   // UNI[6500] := 16#78A3;
   // UNI[6501] := 16#78B2;
   // UNI[6502] := 16#78B9;
   // UNI[6503] := 16#78A5;
   // UNI[6504] := 16#78D4;
   // UNI[6505] := 16#78D9;
   // UNI[6506] := 16#78C9;
   // UNI[6507] := 16#78EC;
   // UNI[6508] := 16#78F2;
   // UNI[6509] := 16#7905;
   // UNI[6510] := 16#78F4;
   // UNI[6511] := 16#7913;
   // UNI[6512] := 16#7924;
   // UNI[6513] := 16#791E;
   // UNI[6514] := 16#7934;
   // UNI[6515] := 16#9F9B;
   // UNI[6516] := 16#9EF9;
   // UNI[6517] := 16#9EFB;
   // UNI[6518] := 16#9EFC;
   // UNI[6519] := 16#76F1;
   // UNI[6520] := 16#7704;
   // UNI[6521] := 16#770D;
   // UNI[6522] := 16#76F9;
   // UNI[6523] := 16#7707;
   // UNI[6524] := 16#7708;
   // UNI[6525] := 16#771A;
   // UNI[6526] := 16#7722;
   // UNI[6527] := 16#7719;
   // UNI[6528] := 16#772D;
   // UNI[6529] := 16#7726;
   // UNI[6530] := 16#7735;
   // UNI[6531] := 16#7738;
   // UNI[6532] := 16#7750;
   // UNI[6533] := 16#7751;
   // UNI[6534] := 16#7747;
   // UNI[6535] := 16#7743;
   // UNI[6536] := 16#775A;
   // UNI[6537] := 16#7768;
   // UNI[6538] := 16#7762;
   // UNI[6539] := 16#7765;
   // UNI[6540] := 16#777F;
   // UNI[6541] := 16#778D;
   // UNI[6542] := 16#777D;
   // UNI[6543] := 16#7780;
   // UNI[6544] := 16#778C;
   // UNI[6545] := 16#7791;
   // UNI[6546] := 16#779F;
   // UNI[6547] := 16#77A0;
   // UNI[6548] := 16#77B0;
   // UNI[6549] := 16#77B5;
   // UNI[6550] := 16#77BD;
   // UNI[6551] := 16#753A;
   // UNI[6552] := 16#7540;
   // UNI[6553] := 16#754E;
   // UNI[6554] := 16#754B;
   // UNI[6555] := 16#7548;
   // UNI[6556] := 16#755B;
   // UNI[6557] := 16#7572;
   // UNI[6558] := 16#7579;
   // UNI[6559] := 16#7583;
   // UNI[6560] := 16#7F58;
   // UNI[6561] := 16#7F61;
   // UNI[6562] := 16#7F5F;
   // UNI[6563] := 16#8A48;
   // UNI[6564] := 16#7F68;
   // UNI[6565] := 16#7F74;
   // UNI[6566] := 16#7F71;
   // UNI[6567] := 16#7F79;
   // UNI[6568] := 16#7F81;
   // UNI[6569] := 16#7F7E;
   // UNI[6570] := 16#76CD;
   // UNI[6571] := 16#76E5;
   // UNI[6572] := 16#8832;
   // UNI[6573] := 16#9485;
   // UNI[6574] := 16#9486;
   // UNI[6575] := 16#9487;
   // UNI[6576] := 16#948B;
   // UNI[6577] := 16#948A;
   // UNI[6578] := 16#948C;
   // UNI[6579] := 16#948D;
   // UNI[6580] := 16#948F;
   // UNI[6581] := 16#9490;
   // UNI[6582] := 16#9494;
   // UNI[6583] := 16#9497;
   // UNI[6584] := 16#9495;
   // UNI[6585] := 16#949A;
   // UNI[6586] := 16#949B;
   // UNI[6587] := 16#949C;
   // UNI[6588] := 16#94A3;
   // UNI[6589] := 16#94A4;
   // UNI[6590] := 16#94AB;
   // UNI[6591] := 16#94AA;
   // UNI[6592] := 16#94AD;
   // UNI[6593] := 16#94AC;
   // UNI[6594] := 16#94AF;
   // UNI[6595] := 16#94B0;
   // UNI[6596] := 16#94B2;
   // UNI[6597] := 16#94B4;
   // UNI[6598] := 16#94B6;
   // UNI[6599] := 16#94B7;
   // UNI[6600] := 16#94B8;
   // UNI[6601] := 16#94B9;
   // UNI[6602] := 16#94BA;
   // UNI[6603] := 16#94BC;
   // UNI[6604] := 16#94BD;
   // UNI[6605] := 16#94BF;
   // UNI[6606] := 16#94C4;
   // UNI[6607] := 16#94C8;
   // UNI[6608] := 16#94C9;
   // UNI[6609] := 16#94CA;
   // UNI[6610] := 16#94CB;
   // UNI[6611] := 16#94CC;
   // UNI[6612] := 16#94CD;
   // UNI[6613] := 16#94CE;
   // UNI[6614] := 16#94D0;
   // UNI[6615] := 16#94D1;
   // UNI[6616] := 16#94D2;
   // UNI[6617] := 16#94D5;
   // UNI[6618] := 16#94D6;
   // UNI[6619] := 16#94D7;
   // UNI[6620] := 16#94D9;
   // UNI[6621] := 16#94D8;
   // UNI[6622] := 16#94DB;
   // UNI[6623] := 16#94DE;
   // UNI[6624] := 16#94DF;
   // UNI[6625] := 16#94E0;
   // UNI[6626] := 16#94E2;
   // UNI[6627] := 16#94E4;
   // UNI[6628] := 16#94E5;
   // UNI[6629] := 16#94E7;
   // UNI[6630] := 16#94E8;
   // UNI[6631] := 16#94EA;
   // UNI[6632] := 16#94E9;
   // UNI[6633] := 16#94EB;
   // UNI[6634] := 16#94EE;
   // UNI[6635] := 16#94EF;
   // UNI[6636] := 16#94F3;
   // UNI[6637] := 16#94F4;
   // UNI[6638] := 16#94F5;
   // UNI[6639] := 16#94F7;
   // UNI[6640] := 16#94F9;
   // UNI[6641] := 16#94FC;
   // UNI[6642] := 16#94FD;
   // UNI[6643] := 16#94FF;
   // UNI[6644] := 16#9503;
   // UNI[6645] := 16#9502;
   // UNI[6646] := 16#9506;
   // UNI[6647] := 16#9507;
   // UNI[6648] := 16#9509;
   // UNI[6649] := 16#950A;
   // UNI[6650] := 16#950D;
   // UNI[6651] := 16#950E;
   // UNI[6652] := 16#950F;
   // UNI[6653] := 16#9512;
   // UNI[6654] := 16#9513;
   // UNI[6655] := 16#9514;
   // UNI[6656] := 16#9515;
   // UNI[6657] := 16#9516;
   // UNI[6658] := 16#9518;
   // UNI[6659] := 16#951B;
   // UNI[6660] := 16#951D;
   // UNI[6661] := 16#951E;
   // UNI[6662] := 16#951F;
   // UNI[6663] := 16#9522;
   // UNI[6664] := 16#952A;
   // UNI[6665] := 16#952B;
   // UNI[6666] := 16#9529;
   // UNI[6667] := 16#952C;
   // UNI[6668] := 16#9531;
   // UNI[6669] := 16#9532;
   // UNI[6670] := 16#9534;
   // UNI[6671] := 16#9536;
   // UNI[6672] := 16#9537;
   // UNI[6673] := 16#9538;
   // UNI[6674] := 16#953C;
   // UNI[6675] := 16#953E;
   // UNI[6676] := 16#953F;
   // UNI[6677] := 16#9542;
   // UNI[6678] := 16#9535;
   // UNI[6679] := 16#9544;
   // UNI[6680] := 16#9545;
   // UNI[6681] := 16#9546;
   // UNI[6682] := 16#9549;
   // UNI[6683] := 16#954C;
   // UNI[6684] := 16#954E;
   // UNI[6685] := 16#954F;
   // UNI[6686] := 16#9552;
   // UNI[6687] := 16#9553;
   // UNI[6688] := 16#9554;
   // UNI[6689] := 16#9556;
   // UNI[6690] := 16#9557;
   // UNI[6691] := 16#9558;
   // UNI[6692] := 16#9559;
   // UNI[6693] := 16#955B;
   // UNI[6694] := 16#955E;
   // UNI[6695] := 16#955F;
   // UNI[6696] := 16#955D;
   // UNI[6697] := 16#9561;
   // UNI[6698] := 16#9562;
   // UNI[6699] := 16#9564;
   // UNI[6700] := 16#9565;
   // UNI[6701] := 16#9566;
   // UNI[6702] := 16#9567;
   // UNI[6703] := 16#9568;
   // UNI[6704] := 16#9569;
   // UNI[6705] := 16#956A;
   // UNI[6706] := 16#956B;
   // UNI[6707] := 16#956C;
   // UNI[6708] := 16#956F;
   // UNI[6709] := 16#9571;
   // UNI[6710] := 16#9572;
   // UNI[6711] := 16#9573;
   // UNI[6712] := 16#953A;
   // UNI[6713] := 16#77E7;
   // UNI[6714] := 16#77EC;
   // UNI[6715] := 16#96C9;
   // UNI[6716] := 16#79D5;
   // UNI[6717] := 16#79ED;
   // UNI[6718] := 16#79E3;
   // UNI[6719] := 16#79EB;
   // UNI[6720] := 16#7A06;
   // UNI[6721] := 16#5D47;
   // UNI[6722] := 16#7A03;
   // UNI[6723] := 16#7A02;
   // UNI[6724] := 16#7A1E;
   // UNI[6725] := 16#7A14;
   // UNI[6726] := 16#7A39;
   // UNI[6727] := 16#7A37;
   // UNI[6728] := 16#7A51;
   // UNI[6729] := 16#9ECF;
   // UNI[6730] := 16#99A5;
   // UNI[6731] := 16#7A70;
   // UNI[6732] := 16#7688;
   // UNI[6733] := 16#768E;
   // UNI[6734] := 16#7693;
   // UNI[6735] := 16#7699;
   // UNI[6736] := 16#76A4;
   // UNI[6737] := 16#74DE;
   // UNI[6738] := 16#74E0;
   // UNI[6739] := 16#752C;
   // UNI[6740] := 16#9E20;
   // UNI[6741] := 16#9E22;
   // UNI[6742] := 16#9E28;
   // UNI[6743] := 16#9E29;
   // UNI[6744] := 16#9E2A;
   // UNI[6745] := 16#9E2B;
   // UNI[6746] := 16#9E2C;
   // UNI[6747] := 16#9E32;
   // UNI[6748] := 16#9E31;
   // UNI[6749] := 16#9E36;
   // UNI[6750] := 16#9E38;
   // UNI[6751] := 16#9E37;
   // UNI[6752] := 16#9E39;
   // UNI[6753] := 16#9E3A;
   // UNI[6754] := 16#9E3E;
   // UNI[6755] := 16#9E41;
   // UNI[6756] := 16#9E42;
   // UNI[6757] := 16#9E44;
   // UNI[6758] := 16#9E46;
   // UNI[6759] := 16#9E47;
   // UNI[6760] := 16#9E48;
   // UNI[6761] := 16#9E49;
   // UNI[6762] := 16#9E4B;
   // UNI[6763] := 16#9E4C;
   // UNI[6764] := 16#9E4E;
   // UNI[6765] := 16#9E51;
   // UNI[6766] := 16#9E55;
   // UNI[6767] := 16#9E57;
   // UNI[6768] := 16#9E5A;
   // UNI[6769] := 16#9E5B;
   // UNI[6770] := 16#9E5C;
   // UNI[6771] := 16#9E5E;
   // UNI[6772] := 16#9E63;
   // UNI[6773] := 16#9E66;
   // UNI[6774] := 16#9E67;
   // UNI[6775] := 16#9E68;
   // UNI[6776] := 16#9E69;
   // UNI[6777] := 16#9E6A;
   // UNI[6778] := 16#9E6B;
   // UNI[6779] := 16#9E6C;
   // UNI[6780] := 16#9E71;
   // UNI[6781] := 16#9E6D;
   // UNI[6782] := 16#9E73;
   // UNI[6783] := 16#7592;
   // UNI[6784] := 16#7594;
   // UNI[6785] := 16#7596;
   // UNI[6786] := 16#75A0;
   // UNI[6787] := 16#759D;
   // UNI[6788] := 16#75AC;
   // UNI[6789] := 16#75A3;
   // UNI[6790] := 16#75B3;
   // UNI[6791] := 16#75B4;
   // UNI[6792] := 16#75B8;
   // UNI[6793] := 16#75C4;
   // UNI[6794] := 16#75B1;
   // UNI[6795] := 16#75B0;
   // UNI[6796] := 16#75C3;
   // UNI[6797] := 16#75C2;
   // UNI[6798] := 16#75D6;
   // UNI[6799] := 16#75CD;
   // UNI[6800] := 16#75E3;
   // UNI[6801] := 16#75E8;
   // UNI[6802] := 16#75E6;
   // UNI[6803] := 16#75E4;
   // UNI[6804] := 16#75EB;
   // UNI[6805] := 16#75E7;
   // UNI[6806] := 16#7603;
   // UNI[6807] := 16#75F1;
   // UNI[6808] := 16#75FC;
   // UNI[6809] := 16#75FF;
   // UNI[6810] := 16#7610;
   // UNI[6811] := 16#7600;
   // UNI[6812] := 16#7605;
   // UNI[6813] := 16#760C;
   // UNI[6814] := 16#7617;
   // UNI[6815] := 16#760A;
   // UNI[6816] := 16#7625;
   // UNI[6817] := 16#7618;
   // UNI[6818] := 16#7615;
   // UNI[6819] := 16#7619;
   // UNI[6820] := 16#761B;
   // UNI[6821] := 16#763C;
   // UNI[6822] := 16#7622;
   // UNI[6823] := 16#7620;
   // UNI[6824] := 16#7640;
   // UNI[6825] := 16#762D;
   // UNI[6826] := 16#7630;
   // UNI[6827] := 16#763F;
   // UNI[6828] := 16#7635;
   // UNI[6829] := 16#7643;
   // UNI[6830] := 16#763E;
   // UNI[6831] := 16#7633;
   // UNI[6832] := 16#764D;
   // UNI[6833] := 16#765E;
   // UNI[6834] := 16#7654;
   // UNI[6835] := 16#765C;
   // UNI[6836] := 16#7656;
   // UNI[6837] := 16#766B;
   // UNI[6838] := 16#766F;
   // UNI[6839] := 16#7FCA;
   // UNI[6840] := 16#7AE6;
   // UNI[6841] := 16#7A78;
   // UNI[6842] := 16#7A79;
   // UNI[6843] := 16#7A80;
   // UNI[6844] := 16#7A86;
   // UNI[6845] := 16#7A88;
   // UNI[6846] := 16#7A95;
   // UNI[6847] := 16#7AA6;
   // UNI[6848] := 16#7AA0;
   // UNI[6849] := 16#7AAC;
   // UNI[6850] := 16#7AA8;
   // UNI[6851] := 16#7AAD;
   // UNI[6852] := 16#7AB3;
   // UNI[6853] := 16#8864;
   // UNI[6854] := 16#8869;
   // UNI[6855] := 16#8872;
   // UNI[6856] := 16#887D;
   // UNI[6857] := 16#887F;
   // UNI[6858] := 16#8882;
   // UNI[6859] := 16#88A2;
   // UNI[6860] := 16#88C6;
   // UNI[6861] := 16#88B7;
   // UNI[6862] := 16#88BC;
   // UNI[6863] := 16#88C9;
   // UNI[6864] := 16#88E2;
   // UNI[6865] := 16#88CE;
   // UNI[6866] := 16#88E3;
   // UNI[6867] := 16#88E5;
   // UNI[6868] := 16#88F1;
   // UNI[6869] := 16#891A;
   // UNI[6870] := 16#88FC;
   // UNI[6871] := 16#88E8;
   // UNI[6872] := 16#88FE;
   // UNI[6873] := 16#88F0;
   // UNI[6874] := 16#8921;
   // UNI[6875] := 16#8919;
   // UNI[6876] := 16#8913;
   // UNI[6877] := 16#891B;
   // UNI[6878] := 16#890A;
   // UNI[6879] := 16#8934;
   // UNI[6880] := 16#892B;
   // UNI[6881] := 16#8936;
   // UNI[6882] := 16#8941;
   // UNI[6883] := 16#8966;
   // UNI[6884] := 16#897B;
   // UNI[6885] := 16#758B;
   // UNI[6886] := 16#80E5;
   // UNI[6887] := 16#76B2;
   // UNI[6888] := 16#76B4;
   // UNI[6889] := 16#77DC;
   // UNI[6890] := 16#8012;
   // UNI[6891] := 16#8014;
   // UNI[6892] := 16#8016;
   // UNI[6893] := 16#801C;
   // UNI[6894] := 16#8020;
   // UNI[6895] := 16#8022;
   // UNI[6896] := 16#8025;
   // UNI[6897] := 16#8026;
   // UNI[6898] := 16#8027;
   // UNI[6899] := 16#8029;
   // UNI[6900] := 16#8028;
   // UNI[6901] := 16#8031;
   // UNI[6902] := 16#800B;
   // UNI[6903] := 16#8035;
   // UNI[6904] := 16#8043;
   // UNI[6905] := 16#8046;
   // UNI[6906] := 16#804D;
   // UNI[6907] := 16#8052;
   // UNI[6908] := 16#8069;
   // UNI[6909] := 16#8071;
   // UNI[6910] := 16#8983;
   // UNI[6911] := 16#9878;
   // UNI[6912] := 16#9880;
   // UNI[6913] := 16#9883;
   // UNI[6914] := 16#9889;
   // UNI[6915] := 16#988C;
   // UNI[6916] := 16#988D;
   // UNI[6917] := 16#988F;
   // UNI[6918] := 16#9894;
   // UNI[6919] := 16#989A;
   // UNI[6920] := 16#989B;
   // UNI[6921] := 16#989E;
   // UNI[6922] := 16#989F;
   // UNI[6923] := 16#98A1;
   // UNI[6924] := 16#98A2;
   // UNI[6925] := 16#98A5;
   // UNI[6926] := 16#98A6;
   // UNI[6927] := 16#864D;
   // UNI[6928] := 16#8654;
   // UNI[6929] := 16#866C;
   // UNI[6930] := 16#866E;
   // UNI[6931] := 16#867F;
   // UNI[6932] := 16#867A;
   // UNI[6933] := 16#867C;
   // UNI[6934] := 16#867B;
   // UNI[6935] := 16#86A8;
   // UNI[6936] := 16#868D;
   // UNI[6937] := 16#868B;
   // UNI[6938] := 16#86AC;
   // UNI[6939] := 16#869D;
   // UNI[6940] := 16#86A7;
   // UNI[6941] := 16#86A3;
   // UNI[6942] := 16#86AA;
   // UNI[6943] := 16#8693;
   // UNI[6944] := 16#86A9;
   // UNI[6945] := 16#86B6;
   // UNI[6946] := 16#86C4;
   // UNI[6947] := 16#86B5;
   // UNI[6948] := 16#86CE;
   // UNI[6949] := 16#86B0;
   // UNI[6950] := 16#86BA;
   // UNI[6951] := 16#86B1;
   // UNI[6952] := 16#86AF;
   // UNI[6953] := 16#86C9;
   // UNI[6954] := 16#86CF;
   // UNI[6955] := 16#86B4;
   // UNI[6956] := 16#86E9;
   // UNI[6957] := 16#86F1;
   // UNI[6958] := 16#86F2;
   // UNI[6959] := 16#86ED;
   // UNI[6960] := 16#86F3;
   // UNI[6961] := 16#86D0;
   // UNI[6962] := 16#8713;
   // UNI[6963] := 16#86DE;
   // UNI[6964] := 16#86F4;
   // UNI[6965] := 16#86DF;
   // UNI[6966] := 16#86D8;
   // UNI[6967] := 16#86D1;
   // UNI[6968] := 16#8703;
   // UNI[6969] := 16#8707;
   // UNI[6970] := 16#86F8;
   // UNI[6971] := 16#8708;
   // UNI[6972] := 16#870A;
   // UNI[6973] := 16#870D;
   // UNI[6974] := 16#8709;
   // UNI[6975] := 16#8723;
   // UNI[6976] := 16#873B;
   // UNI[6977] := 16#871E;
   // UNI[6978] := 16#8725;
   // UNI[6979] := 16#872E;
   // UNI[6980] := 16#871A;
   // UNI[6981] := 16#873E;
   // UNI[6982] := 16#8748;
   // UNI[6983] := 16#8734;
   // UNI[6984] := 16#8731;
   // UNI[6985] := 16#8729;
   // UNI[6986] := 16#8737;
   // UNI[6987] := 16#873F;
   // UNI[6988] := 16#8782;
   // UNI[6989] := 16#8722;
   // UNI[6990] := 16#877D;
   // UNI[6991] := 16#877E;
   // UNI[6992] := 16#877B;
   // UNI[6993] := 16#8760;
   // UNI[6994] := 16#8770;
   // UNI[6995] := 16#874C;
   // UNI[6996] := 16#876E;
   // UNI[6997] := 16#878B;
   // UNI[6998] := 16#8753;
   // UNI[6999] := 16#8763;
   // UNI[7000] := 16#877C;
   // UNI[7001] := 16#8764;
   // UNI[7002] := 16#8759;
   // UNI[7003] := 16#8765;
   // UNI[7004] := 16#8793;
   // UNI[7005] := 16#87AF;
   // UNI[7006] := 16#87A8;
   // UNI[7007] := 16#87D2;
   // UNI[7008] := 16#87C6;
   // UNI[7009] := 16#8788;
   // UNI[7010] := 16#8785;
   // UNI[7011] := 16#87AD;
   // UNI[7012] := 16#8797;
   // UNI[7013] := 16#8783;
   // UNI[7014] := 16#87AB;
   // UNI[7015] := 16#87E5;
   // UNI[7016] := 16#87AC;
   // UNI[7017] := 16#87B5;
   // UNI[7018] := 16#87B3;
   // UNI[7019] := 16#87CB;
   // UNI[7020] := 16#87D3;
   // UNI[7021] := 16#87BD;
   // UNI[7022] := 16#87D1;
   // UNI[7023] := 16#87C0;
   // UNI[7024] := 16#87CA;
   // UNI[7025] := 16#87DB;
   // UNI[7026] := 16#87EA;
   // UNI[7027] := 16#87E0;
   // UNI[7028] := 16#87EE;
   // UNI[7029] := 16#8816;
   // UNI[7030] := 16#8813;
   // UNI[7031] := 16#87FE;
   // UNI[7032] := 16#880A;
   // UNI[7033] := 16#881B;
   // UNI[7034] := 16#8821;
   // UNI[7035] := 16#8839;
   // UNI[7036] := 16#883C;
   // UNI[7037] := 16#7F36;
   // UNI[7038] := 16#7F42;
   // UNI[7039] := 16#7F44;
   // UNI[7040] := 16#7F45;
   // UNI[7041] := 16#8210;
   // UNI[7042] := 16#7AFA;
   // UNI[7043] := 16#7AFD;
   // UNI[7044] := 16#7B08;
   // UNI[7045] := 16#7B03;
   // UNI[7046] := 16#7B04;
   // UNI[7047] := 16#7B15;
   // UNI[7048] := 16#7B0A;
   // UNI[7049] := 16#7B2B;
   // UNI[7050] := 16#7B0F;
   // UNI[7051] := 16#7B47;
   // UNI[7052] := 16#7B38;
   // UNI[7053] := 16#7B2A;
   // UNI[7054] := 16#7B19;
   // UNI[7055] := 16#7B2E;
   // UNI[7056] := 16#7B31;
   // UNI[7057] := 16#7B20;
   // UNI[7058] := 16#7B25;
   // UNI[7059] := 16#7B24;
   // UNI[7060] := 16#7B33;
   // UNI[7061] := 16#7B3E;
   // UNI[7062] := 16#7B1E;
   // UNI[7063] := 16#7B58;
   // UNI[7064] := 16#7B5A;
   // UNI[7065] := 16#7B45;
   // UNI[7066] := 16#7B75;
   // UNI[7067] := 16#7B4C;
   // UNI[7068] := 16#7B5D;
   // UNI[7069] := 16#7B60;
   // UNI[7070] := 16#7B6E;
   // UNI[7071] := 16#7B7B;
   // UNI[7072] := 16#7B62;
   // UNI[7073] := 16#7B72;
   // UNI[7074] := 16#7B71;
   // UNI[7075] := 16#7B90;
   // UNI[7076] := 16#7BA6;
   // UNI[7077] := 16#7BA7;
   // UNI[7078] := 16#7BB8;
   // UNI[7079] := 16#7BAC;
   // UNI[7080] := 16#7B9D;
   // UNI[7081] := 16#7BA8;
   // UNI[7082] := 16#7B85;
   // UNI[7083] := 16#7BAA;
   // UNI[7084] := 16#7B9C;
   // UNI[7085] := 16#7BA2;
   // UNI[7086] := 16#7BAB;
   // UNI[7087] := 16#7BB4;
   // UNI[7088] := 16#7BD1;
   // UNI[7089] := 16#7BC1;
   // UNI[7090] := 16#7BCC;
   // UNI[7091] := 16#7BDD;
   // UNI[7092] := 16#7BDA;
   // UNI[7093] := 16#7BE5;
   // UNI[7094] := 16#7BE6;
   // UNI[7095] := 16#7BEA;
   // UNI[7096] := 16#7C0C;
   // UNI[7097] := 16#7BFE;
   // UNI[7098] := 16#7BFC;
   // UNI[7099] := 16#7C0F;
   // UNI[7100] := 16#7C16;
   // UNI[7101] := 16#7C0B;
   // UNI[7102] := 16#7C1F;
   // UNI[7103] := 16#7C2A;
   // UNI[7104] := 16#7C26;
   // UNI[7105] := 16#7C38;
   // UNI[7106] := 16#7C41;
   // UNI[7107] := 16#7C40;
   // UNI[7108] := 16#81FE;
   // UNI[7109] := 16#8201;
   // UNI[7110] := 16#8202;
   // UNI[7111] := 16#8204;
   // UNI[7112] := 16#81EC;
   // UNI[7113] := 16#8844;
   // UNI[7114] := 16#8221;
   // UNI[7115] := 16#8222;
   // UNI[7116] := 16#8223;
   // UNI[7117] := 16#822D;
   // UNI[7118] := 16#822F;
   // UNI[7119] := 16#8228;
   // UNI[7120] := 16#822B;
   // UNI[7121] := 16#8238;
   // UNI[7122] := 16#823B;
   // UNI[7123] := 16#8233;
   // UNI[7124] := 16#8234;
   // UNI[7125] := 16#823E;
   // UNI[7126] := 16#8244;
   // UNI[7127] := 16#8249;
   // UNI[7128] := 16#824B;
   // UNI[7129] := 16#824F;
   // UNI[7130] := 16#825A;
   // UNI[7131] := 16#825F;
   // UNI[7132] := 16#8268;
   // UNI[7133] := 16#887E;
   // UNI[7134] := 16#8885;
   // UNI[7135] := 16#8888;
   // UNI[7136] := 16#88D8;
   // UNI[7137] := 16#88DF;
   // UNI[7138] := 16#895E;
   // UNI[7139] := 16#7F9D;
   // UNI[7140] := 16#7F9F;
   // UNI[7141] := 16#7FA7;
   // UNI[7142] := 16#7FAF;
   // UNI[7143] := 16#7FB0;
   // UNI[7144] := 16#7FB2;
   // UNI[7145] := 16#7C7C;
   // UNI[7146] := 16#6549;
   // UNI[7147] := 16#7C91;
   // UNI[7148] := 16#7C9D;
   // UNI[7149] := 16#7C9C;
   // UNI[7150] := 16#7C9E;
   // UNI[7151] := 16#7CA2;
   // UNI[7152] := 16#7CB2;
   // UNI[7153] := 16#7CBC;
   // UNI[7154] := 16#7CBD;
   // UNI[7155] := 16#7CC1;
   // UNI[7156] := 16#7CC7;
   // UNI[7157] := 16#7CCC;
   // UNI[7158] := 16#7CCD;
   // UNI[7159] := 16#7CC8;
   // UNI[7160] := 16#7CC5;
   // UNI[7161] := 16#7CD7;
   // UNI[7162] := 16#7CE8;
   // UNI[7163] := 16#826E;
   // UNI[7164] := 16#66A8;
   // UNI[7165] := 16#7FBF;
   // UNI[7166] := 16#7FCE;
   // UNI[7167] := 16#7FD5;
   // UNI[7168] := 16#7FE5;
   // UNI[7169] := 16#7FE1;
   // UNI[7170] := 16#7FE6;
   // UNI[7171] := 16#7FE9;
   // UNI[7172] := 16#7FEE;
   // UNI[7173] := 16#7FF3;
   // UNI[7174] := 16#7CF8;
   // UNI[7175] := 16#7D77;
   // UNI[7176] := 16#7DA6;
   // UNI[7177] := 16#7DAE;
   // UNI[7178] := 16#7E47;
   // UNI[7179] := 16#7E9B;
   // UNI[7180] := 16#9EB8;
   // UNI[7181] := 16#9EB4;
   // UNI[7182] := 16#8D73;
   // UNI[7183] := 16#8D84;
   // UNI[7184] := 16#8D94;
   // UNI[7185] := 16#8D91;
   // UNI[7186] := 16#8DB1;
   // UNI[7187] := 16#8D67;
   // UNI[7188] := 16#8D6D;
   // UNI[7189] := 16#8C47;
   // UNI[7190] := 16#8C49;
   // UNI[7191] := 16#914A;
   // UNI[7192] := 16#9150;
   // UNI[7193] := 16#914E;
   // UNI[7194] := 16#914F;
   // UNI[7195] := 16#9164;
   // UNI[7196] := 16#9162;
   // UNI[7197] := 16#9161;
   // UNI[7198] := 16#9170;
   // UNI[7199] := 16#9169;
   // UNI[7200] := 16#916F;
   // UNI[7201] := 16#917D;
   // UNI[7202] := 16#917E;
   // UNI[7203] := 16#9172;
   // UNI[7204] := 16#9174;
   // UNI[7205] := 16#9179;
   // UNI[7206] := 16#918C;
   // UNI[7207] := 16#9185;
   // UNI[7208] := 16#9190;
   // UNI[7209] := 16#918D;
   // UNI[7210] := 16#9191;
   // UNI[7211] := 16#91A2;
   // UNI[7212] := 16#91A3;
   // UNI[7213] := 16#91AA;
   // UNI[7214] := 16#91AD;
   // UNI[7215] := 16#91AE;
   // UNI[7216] := 16#91AF;
   // UNI[7217] := 16#91B5;
   // UNI[7218] := 16#91B4;
   // UNI[7219] := 16#91BA;
   // UNI[7220] := 16#8C55;
   // UNI[7221] := 16#9E7E;
   // UNI[7222] := 16#8DB8;
   // UNI[7223] := 16#8DEB;
   // UNI[7224] := 16#8E05;
   // UNI[7225] := 16#8E59;
   // UNI[7226] := 16#8E69;
   // UNI[7227] := 16#8DB5;
   // UNI[7228] := 16#8DBF;
   // UNI[7229] := 16#8DBC;
   // UNI[7230] := 16#8DBA;
   // UNI[7231] := 16#8DC4;
   // UNI[7232] := 16#8DD6;
   // UNI[7233] := 16#8DD7;
   // UNI[7234] := 16#8DDA;
   // UNI[7235] := 16#8DDE;
   // UNI[7236] := 16#8DCE;
   // UNI[7237] := 16#8DCF;
   // UNI[7238] := 16#8DDB;
   // UNI[7239] := 16#8DC6;
   // UNI[7240] := 16#8DEC;
   // UNI[7241] := 16#8DF7;
   // UNI[7242] := 16#8DF8;
   // UNI[7243] := 16#8DE3;
   // UNI[7244] := 16#8DF9;
   // UNI[7245] := 16#8DFB;
   // UNI[7246] := 16#8DE4;
   // UNI[7247] := 16#8E09;
   // UNI[7248] := 16#8DFD;
   // UNI[7249] := 16#8E14;
   // UNI[7250] := 16#8E1D;
   // UNI[7251] := 16#8E1F;
   // UNI[7252] := 16#8E2C;
   // UNI[7253] := 16#8E2E;
   // UNI[7254] := 16#8E23;
   // UNI[7255] := 16#8E2F;
   // UNI[7256] := 16#8E3A;
   // UNI[7257] := 16#8E40;
   // UNI[7258] := 16#8E39;
   // UNI[7259] := 16#8E35;
   // UNI[7260] := 16#8E3D;
   // UNI[7261] := 16#8E31;
   // UNI[7262] := 16#8E49;
   // UNI[7263] := 16#8E41;
   // UNI[7264] := 16#8E42;
   // UNI[7265] := 16#8E51;
   // UNI[7266] := 16#8E52;
   // UNI[7267] := 16#8E4A;
   // UNI[7268] := 16#8E70;
   // UNI[7269] := 16#8E76;
   // UNI[7270] := 16#8E7C;
   // UNI[7271] := 16#8E6F;
   // UNI[7272] := 16#8E74;
   // UNI[7273] := 16#8E85;
   // UNI[7274] := 16#8E8F;
   // UNI[7275] := 16#8E94;
   // UNI[7276] := 16#8E90;
   // UNI[7277] := 16#8E9C;
   // UNI[7278] := 16#8E9E;
   // UNI[7279] := 16#8C78;
   // UNI[7280] := 16#8C82;
   // UNI[7281] := 16#8C8A;
   // UNI[7282] := 16#8C85;
   // UNI[7283] := 16#8C98;
   // UNI[7284] := 16#8C94;
   // UNI[7285] := 16#659B;
   // UNI[7286] := 16#89D6;
   // UNI[7287] := 16#89DE;
   // UNI[7288] := 16#89DA;
   // UNI[7289] := 16#89DC;
   // UNI[7290] := 16#89E5;
   // UNI[7291] := 16#89EB;
   // UNI[7292] := 16#89EF;
   // UNI[7293] := 16#8A3E;
   // UNI[7294] := 16#8B26;
   // UNI[7295] := 16#9753;
   // UNI[7296] := 16#96E9;
   // UNI[7297] := 16#96F3;
   // UNI[7298] := 16#96EF;
   // UNI[7299] := 16#9706;
   // UNI[7300] := 16#9701;
   // UNI[7301] := 16#9708;
   // UNI[7302] := 16#970F;
   // UNI[7303] := 16#970E;
   // UNI[7304] := 16#972A;
   // UNI[7305] := 16#972D;
   // UNI[7306] := 16#9730;
   // UNI[7307] := 16#973E;
   // UNI[7308] := 16#9F80;
   // UNI[7309] := 16#9F83;
   // UNI[7310] := 16#9F85;
   // UNI[7311] := 16#9F86;
   // UNI[7312] := 16#9F87;
   // UNI[7313] := 16#9F88;
   // UNI[7314] := 16#9F89;
   // UNI[7315] := 16#9F8A;
   // UNI[7316] := 16#9F8C;
   // UNI[7317] := 16#9EFE;
   // UNI[7318] := 16#9F0B;
   // UNI[7319] := 16#9F0D;
   // UNI[7320] := 16#96B9;
   // UNI[7321] := 16#96BC;
   // UNI[7322] := 16#96BD;
   // UNI[7323] := 16#96CE;
   // UNI[7324] := 16#96D2;
   // UNI[7325] := 16#77BF;
   // UNI[7326] := 16#96E0;
   // UNI[7327] := 16#928E;
   // UNI[7328] := 16#92AE;
   // UNI[7329] := 16#92C8;
   // UNI[7330] := 16#933E;
   // UNI[7331] := 16#936A;
   // UNI[7332] := 16#93CA;
   // UNI[7333] := 16#938F;
   // UNI[7334] := 16#943E;
   // UNI[7335] := 16#946B;
   // UNI[7336] := 16#9C7F;
   // UNI[7337] := 16#9C82;
   // UNI[7338] := 16#9C85;
   // UNI[7339] := 16#9C86;
   // UNI[7340] := 16#9C87;
   // UNI[7341] := 16#9C88;
   // UNI[7342] := 16#7A23;
   // UNI[7343] := 16#9C8B;
   // UNI[7344] := 16#9C8E;
   // UNI[7345] := 16#9C90;
   // UNI[7346] := 16#9C91;
   // UNI[7347] := 16#9C92;
   // UNI[7348] := 16#9C94;
   // UNI[7349] := 16#9C95;
   // UNI[7350] := 16#9C9A;
   // UNI[7351] := 16#9C9B;
   // UNI[7352] := 16#9C9E;
   // UNI[7353] := 16#9C9F;
   // UNI[7354] := 16#9CA0;
   // UNI[7355] := 16#9CA1;
   // UNI[7356] := 16#9CA2;
   // UNI[7357] := 16#9CA3;
   // UNI[7358] := 16#9CA5;
   // UNI[7359] := 16#9CA6;
   // UNI[7360] := 16#9CA7;
   // UNI[7361] := 16#9CA8;
   // UNI[7362] := 16#9CA9;
   // UNI[7363] := 16#9CAB;
   // UNI[7364] := 16#9CAD;
   // UNI[7365] := 16#9CAE;
   // UNI[7366] := 16#9CB0;
   // UNI[7367] := 16#9CB1;
   // UNI[7368] := 16#9CB2;
   // UNI[7369] := 16#9CB3;
   // UNI[7370] := 16#9CB4;
   // UNI[7371] := 16#9CB5;
   // UNI[7372] := 16#9CB6;
   // UNI[7373] := 16#9CB7;
   // UNI[7374] := 16#9CBA;
   // UNI[7375] := 16#9CBB;
   // UNI[7376] := 16#9CBC;
   // UNI[7377] := 16#9CBD;
   // UNI[7378] := 16#9CC4;
   // UNI[7379] := 16#9CC5;
   // UNI[7380] := 16#9CC6;
   // UNI[7381] := 16#9CC7;
   // UNI[7382] := 16#9CCA;
   // UNI[7383] := 16#9CCB;
   // UNI[7384] := 16#9CCC;
   // UNI[7385] := 16#9CCD;
   // UNI[7386] := 16#9CCE;
   // UNI[7387] := 16#9CCF;
   // UNI[7388] := 16#9CD0;
   // UNI[7389] := 16#9CD3;
   // UNI[7390] := 16#9CD4;
   // UNI[7391] := 16#9CD5;
   // UNI[7392] := 16#9CD7;
   // UNI[7393] := 16#9CD8;
   // UNI[7394] := 16#9CD9;
   // UNI[7395] := 16#9CDC;
   // UNI[7396] := 16#9CDD;
   // UNI[7397] := 16#9CDF;
   // UNI[7398] := 16#9CE2;
   // UNI[7399] := 16#977C;
   // UNI[7400] := 16#9785;
   // UNI[7401] := 16#9791;
   // UNI[7402] := 16#9792;
   // UNI[7403] := 16#9794;
   // UNI[7404] := 16#97AF;
   // UNI[7405] := 16#97AB;
   // UNI[7406] := 16#97A3;
   // UNI[7407] := 16#97B2;
   // UNI[7408] := 16#97B4;
   // UNI[7409] := 16#9AB1;
   // UNI[7410] := 16#9AB0;
   // UNI[7411] := 16#9AB7;
   // UNI[7412] := 16#9E58;
   // UNI[7413] := 16#9AB6;
   // UNI[7414] := 16#9ABA;
   // UNI[7415] := 16#9ABC;
   // UNI[7416] := 16#9AC1;
   // UNI[7417] := 16#9AC0;
   // UNI[7418] := 16#9AC5;
   // UNI[7419] := 16#9AC2;
   // UNI[7420] := 16#9ACB;
   // UNI[7421] := 16#9ACC;
   // UNI[7422] := 16#9AD1;
   // UNI[7423] := 16#9B45;
   // UNI[7424] := 16#9B43;
   // UNI[7425] := 16#9B47;
   // UNI[7426] := 16#9B49;
   // UNI[7427] := 16#9B48;
   // UNI[7428] := 16#9B4D;
   // UNI[7429] := 16#9B51;
   // UNI[7430] := 16#98E8;
   // UNI[7431] := 16#990D;
   // UNI[7432] := 16#992E;
   // UNI[7433] := 16#9955;
   // UNI[7434] := 16#9954;
   // UNI[7435] := 16#9ADF;
   // UNI[7436] := 16#9AE1;
   // UNI[7437] := 16#9AE6;
   // UNI[7438] := 16#9AEF;
   // UNI[7439] := 16#9AEB;
   // UNI[7440] := 16#9AFB;
   // UNI[7441] := 16#9AED;
   // UNI[7442] := 16#9AF9;
   // UNI[7443] := 16#9B08;
   // UNI[7444] := 16#9B0F;
   // UNI[7445] := 16#9B13;
   // UNI[7446] := 16#9B1F;
   // UNI[7447] := 16#9B23;
   // UNI[7448] := 16#9EBD;
   // UNI[7449] := 16#9EBE;
   // UNI[7450] := 16#7E3B;
   // UNI[7451] := 16#9E82;
   // UNI[7452] := 16#9E87;
   // UNI[7453] := 16#9E88;
   // UNI[7454] := 16#9E8B;
   // UNI[7455] := 16#9E92;
   // UNI[7456] := 16#93D6;
   // UNI[7457] := 16#9E9D;
   // UNI[7458] := 16#9E9F;
   // UNI[7459] := 16#9EDB;
   // UNI[7460] := 16#9EDC;
   // UNI[7461] := 16#9EDD;
   // UNI[7462] := 16#9EE0;
   // UNI[7463] := 16#9EDF;
   // UNI[7464] := 16#9EE2;
   // UNI[7465] := 16#9EE9;
   // UNI[7466] := 16#9EE7;
   // UNI[7467] := 16#9EE5;
   // UNI[7468] := 16#9EEA;
   // UNI[7469] := 16#9EEF;
   // UNI[7470] := 16#9F22;
   // UNI[7471] := 16#9F2C;
   // UNI[7472] := 16#9F2F;
   // UNI[7473] := 16#9F39;
   // UNI[7474] := 16#9F37;
   // UNI[7475] := 16#9F3D;
   // UNI[7476] := 16#9F3E;
   // UNI[7477] := 16#9F44;
   // UNI[7478] := 0;
   // UNI[7479] := 0;
BEGIN
   IF #GB2312 < 16#0080 THEN
       #UNICODE := #GB2312;
   ELSE
       #hi := 7480;
       #li := 0;
       FOR #j := 0 TO 13 BY 1 DO
           #i := #li + (#hi - #li) / 2;
           IF #GB2312 = #GB2[#i] THEN
               #UNICODE := #UNI[#i];
               EXIT;
           END_IF;
           IF #GB2312 > #GB2[#i] THEN
               #li := #i;
           ELSE
               #hi := #i;
           END_IF;
       END_FOR;
   END_IF;
END_FUNCTION_BLOCK

// ===== library: MasterCopy "GBK_TO_UNI" =====

// folder: FB/UNICODE_FB

FUNCTION_BLOCK "GBK_TO_UNI"   // FB2, SCL
{ S7_Optimized_Access := 'TRUE' }
VERSION : 0.1
   VAR_INPUT
      GBK : Word;
   END_VAR
   VAR_OUTPUT
      UNICODE : Word;
   END_VAR
   VAR
      GBK_TO_UNICODE : Array[0..43592] of Word;
   END_VAR
   VAR_TEMP
      i : UDInt;
      j : UDInt;
      li : UDInt;
      hi : UDInt;
   END_VAR
   // GBK_TO_UNICODE[0] := 16#0080;
   // GBK_TO_UNICODE[1] := 16#20AC;
   // GBK_TO_UNICODE[2] := 16#8140;
   // GBK_TO_UNICODE[3] := 16#4E02;
   // GBK_TO_UNICODE[4] := 16#8141;
   // GBK_TO_UNICODE[5] := 16#4E04;
   // GBK_TO_UNICODE[6] := 16#8142;
   // GBK_TO_UNICODE[7] := 16#4E05;
   // GBK_TO_UNICODE[8] := 16#8143;
   // GBK_TO_UNICODE[9] := 16#4E06;
   // GBK_TO_UNICODE[10] := 16#8144;
   // GBK_TO_UNICODE[11] := 16#4E0F;
   // GBK_TO_UNICODE[12] := 16#8145;
   // GBK_TO_UNICODE[13] := 16#4E12;
   // GBK_TO_UNICODE[14] := 16#8146;
   // GBK_TO_UNICODE[15] := 16#4E17;
   // GBK_TO_UNICODE[16] := 16#8147;
   // GBK_TO_UNICODE[17] := 16#4E1F;
   // GBK_TO_UNICODE[18] := 16#8148;
   // GBK_TO_UNICODE[19] := 16#4E20;
   // GBK_TO_UNICODE[20] := 16#8149;
   // GBK_TO_UNICODE[21] := 16#4E21;
   // GBK_TO_UNICODE[22] := 16#814A;
   // GBK_TO_UNICODE[23] := 16#4E23;
   // GBK_TO_UNICODE[24] := 16#814B;
   // GBK_TO_UNICODE[25] := 16#4E26;
   // GBK_TO_UNICODE[26] := 16#814C;
   // GBK_TO_UNICODE[27] := 16#4E29;
   // GBK_TO_UNICODE[28] := 16#814D;
   // GBK_TO_UNICODE[29] := 16#4E2E;
   // GBK_TO_UNICODE[30] := 16#814E;
   // GBK_TO_UNICODE[31] := 16#4E2F;
   // GBK_TO_UNICODE[32] := 16#814F;
   // GBK_TO_UNICODE[33] := 16#4E31;
   // GBK_TO_UNICODE[34] := 16#8150;
   // GBK_TO_UNICODE[35] := 16#4E33;
   // GBK_TO_UNICODE[36] := 16#8151;
   // GBK_TO_UNICODE[37] := 16#4E35;
   // GBK_TO_UNICODE[38] := 16#8152;
   // GBK_TO_UNICODE[39] := 16#4E37;
   // GBK_TO_UNICODE[40] := 16#8153;
   // GBK_TO_UNICODE[41] := 16#4E3C;
   // GBK_TO_UNICODE[42] := 16#8154;
   // GBK_TO_UNICODE[43] := 16#4E40;
   // GBK_TO_UNICODE[44] := 16#8155;
   // GBK_TO_UNICODE[45] := 16#4E41;
   // GBK_TO_UNICODE[46] := 16#8156;
   // GBK_TO_UNICODE[47] := 16#4E42;
   // GBK_TO_UNICODE[48] := 16#8157;
   // GBK_TO_UNICODE[49] := 16#4E44;
   // GBK_TO_UNICODE[50] := 16#8158;
   // GBK_TO_UNICODE[51] := 16#4E46;
   // GBK_TO_UNICODE[52] := 16#8159;
   // GBK_TO_UNICODE[53] := 16#4E4A;
   // GBK_TO_UNICODE[54] := 16#815A;
   // GBK_TO_UNICODE[55] := 16#4E51;
   // GBK_TO_UNICODE[56] := 16#815B;
   // GBK_TO_UNICODE[57] := 16#4E55;
   // GBK_TO_UNICODE[58] := 16#815C;
   // GBK_TO_UNICODE[59] := 16#4E57;
   // GBK_TO_UNICODE[60] := 16#815D;
   // GBK_TO_UNICODE[61] := 16#4E5A;
   // GBK_TO_UNICODE[62] := 16#815E;
   // GBK_TO_UNICODE[63] := 16#4E5B;
   // GBK_TO_UNICODE[64] := 16#815F;
   // GBK_TO_UNICODE[65] := 16#4E62;
   // GBK_TO_UNICODE[66] := 16#8160;
   // GBK_TO_UNICODE[67] := 16#4E63;
   // GBK_TO_UNICODE[68] := 16#8161;
   // GBK_TO_UNICODE[69] := 16#4E64;
   // GBK_TO_UNICODE[70] := 16#8162;
   // GBK_TO_UNICODE[71] := 16#4E65;
   // GBK_TO_UNICODE[72] := 16#8163;
   // GBK_TO_UNICODE[73] := 16#4E67;
   // GBK_TO_UNICODE[74] := 16#8164;
   // GBK_TO_UNICODE[75] := 16#4E68;
   // GBK_TO_UNICODE[76] := 16#8165;
   // GBK_TO_UNICODE[77] := 16#4E6A;
   // GBK_TO_UNICODE[78] := 16#8166;
   // GBK_TO_UNICODE[79] := 16#4E6B;
   // GBK_TO_UNICODE[80] := 16#8167;
   // GBK_TO_UNICODE[81] := 16#4E6C;
   // GBK_TO_UNICODE[82] := 16#8168;
   // GBK_TO_UNICODE[83] := 16#4E6D;
   // GBK_TO_UNICODE[84] := 16#8169;
   // GBK_TO_UNICODE[85] := 16#4E6E;
   // GBK_TO_UNICODE[86] := 16#816A;
   // GBK_TO_UNICODE[87] := 16#4E6F;
   // GBK_TO_UNICODE[88] := 16#816B;
   // GBK_TO_UNICODE[89] := 16#4E72;
   // GBK_TO_UNICODE[90] := 16#816C;
   // GBK_TO_UNICODE[91] := 16#4E74;
   // GBK_TO_UNICODE[92] := 16#816D;
   // GBK_TO_UNICODE[93] := 16#4E75;
   // GBK_TO_UNICODE[94] := 16#816E;
   // GBK_TO_UNICODE[95] := 16#4E76;
   // GBK_TO_UNICODE[96] := 16#816F;
   // GBK_TO_UNICODE[97] := 16#4E77;
   // GBK_TO_UNICODE[98] := 16#8170;
   // GBK_TO_UNICODE[99] := 16#4E78;
   // GBK_TO_UNICODE[100] := 16#8171;
   // GBK_TO_UNICODE[101] := 16#4E79;
   // GBK_TO_UNICODE[102] := 16#8172;
   // GBK_TO_UNICODE[103] := 16#4E7A;
   // GBK_TO_UNICODE[104] := 16#8173;
   // GBK_TO_UNICODE[105] := 16#4E7B;
   // GBK_TO_UNICODE[106] := 16#8174;
   // GBK_TO_UNICODE[107] := 16#4E7C;
   // GBK_TO_UNICODE[108] := 16#8175;
   // GBK_TO_UNICODE[109] := 16#4E7D;
   // GBK_TO_UNICODE[110] := 16#8176;
   // GBK_TO_UNICODE[111] := 16#4E7F;
   // GBK_TO_UNICODE[112] := 16#8177;
   // GBK_TO_UNICODE[113] := 16#4E80;
   // GBK_TO_UNICODE[114] := 16#8178;
   // GBK_TO_UNICODE[115] := 16#4E81;
   // GBK_TO_UNICODE[116] := 16#8179;
   // GBK_TO_UNICODE[117] := 16#4E82;
   // GBK_TO_UNICODE[118] := 16#817A;
   // GBK_TO_UNICODE[119] := 16#4E83;
   // GBK_TO_UNICODE[120] := 16#817B;
   // GBK_TO_UNICODE[121] := 16#4E84;
   // GBK_TO_UNICODE[122] := 16#817C;
   // GBK_TO_UNICODE[123] := 16#4E85;
   // GBK_TO_UNICODE[124] := 16#817D;
   // GBK_TO_UNICODE[125] := 16#4E87;
   // GBK_TO_UNICODE[126] := 16#817E;
   // GBK_TO_UNICODE[127] := 16#4E8A;
   // GBK_TO_UNICODE[128] := 16#8180;
   // GBK_TO_UNICODE[129] := 16#4E90;
   // GBK_TO_UNICODE[130] := 16#8181;
   // GBK_TO_UNICODE[131] := 16#4E96;
   // GBK_TO_UNICODE[132] := 16#8182;
   // GBK_TO_UNICODE[133] := 16#4E97;
   // GBK_TO_UNICODE[134] := 16#8183;
   // GBK_TO_UNICODE[135] := 16#4E99;
   // GBK_TO_UNICODE[136] := 16#8184;
   // GBK_TO_UNICODE[137] := 16#4E9C;
   // GBK_TO_UNICODE[138] := 16#8185;
   // GBK_TO_UNICODE[139] := 16#4E9D;
   // GBK_TO_UNICODE[140] := 16#8186;
   // GBK_TO_UNICODE[141] := 16#4E9E;
   // GBK_TO_UNICODE[142] := 16#8187;
   // GBK_TO_UNICODE[143] := 16#4EA3;
   // GBK_TO_UNICODE[144] := 16#8188;
   // GBK_TO_UNICODE[145] := 16#4EAA;
   // GBK_TO_UNICODE[146] := 16#8189;
   // GBK_TO_UNICODE[147] := 16#4EAF;
   // GBK_TO_UNICODE[148] := 16#818A;
   // GBK_TO_UNICODE[149] := 16#4EB0;
   // GBK_TO_UNICODE[150] := 16#818B;
   // GBK_TO_UNICODE[151] := 16#4EB1;
   // GBK_TO_UNICODE[152] := 16#818C;
   // GBK_TO_UNICODE[153] := 16#4EB4;
   // GBK_TO_UNICODE[154] := 16#818D;
   // GBK_TO_UNICODE[155] := 16#4EB6;
   // GBK_TO_UNICODE[156] := 16#818E;
   // GBK_TO_UNICODE[157] := 16#4EB7;
   // GBK_TO_UNICODE[158] := 16#818F;
   // GBK_TO_UNICODE[159] := 16#4EB8;
   // GBK_TO_UNICODE[160] := 16#8190;
   // GBK_TO_UNICODE[161] := 16#4EB9;
   // GBK_TO_UNICODE[162] := 16#8191;
   // GBK_TO_UNICODE[163] := 16#4EBC;
   // GBK_TO_UNICODE[164] := 16#8192;
   // GBK_TO_UNICODE[165] := 16#4EBD;
   // GBK_TO_UNICODE[166] := 16#8193;
   // GBK_TO_UNICODE[167] := 16#4EBE;
   // GBK_TO_UNICODE[168] := 16#8194;
   // GBK_TO_UNICODE[169] := 16#4EC8;
   // GBK_TO_UNICODE[170] := 16#8195;
   // GBK_TO_UNICODE[171] := 16#4ECC;
   // GBK_TO_UNICODE[172] := 16#8196;
   // GBK_TO_UNICODE[173] := 16#4ECF;
   // GBK_TO_UNICODE[174] := 16#8197;
   // GBK_TO_UNICODE[175] := 16#4ED0;
   // GBK_TO_UNICODE[176] := 16#8198;
   // GBK_TO_UNICODE[177] := 16#4ED2;
   // GBK_TO_UNICODE[178] := 16#8199;
   // GBK_TO_UNICODE[179] := 16#4EDA;
   // GBK_TO_UNICODE[180] := 16#819A;
   // GBK_TO_UNICODE[181] := 16#4EDB;
   // GBK_TO_UNICODE[182] := 16#819B;
   // GBK_TO_UNICODE[183] := 16#4EDC;
   // GBK_TO_UNICODE[184] := 16#819C;
   // GBK_TO_UNICODE[185] := 16#4EE0;
   // GBK_TO_UNICODE[186] := 16#819D;
   // GBK_TO_UNICODE[187] := 16#4EE2;
   // GBK_TO_UNICODE[188] := 16#819E;
   // GBK_TO_UNICODE[189] := 16#4EE6;
   // GBK_TO_UNICODE[190] := 16#819F;
   // GBK_TO_UNICODE[191] := 16#4EE7;
   // GBK_TO_UNICODE[192] := 16#81A0;
   // GBK_TO_UNICODE[193] := 16#4EE9;
   // GBK_TO_UNICODE[194] := 16#81A1;
   // GBK_TO_UNICODE[195] := 16#4EED;
   // GBK_TO_UNICODE[196] := 16#81A2;
   // GBK_TO_UNICODE[197] := 16#4EEE;
   // GBK_TO_UNICODE[198] := 16#81A3;
   // GBK_TO_UNICODE[199] := 16#4EEF;
   // GBK_TO_UNICODE[200] := 16#81A4;
   // GBK_TO_UNICODE[201] := 16#4EF1;
   // GBK_TO_UNICODE[202] := 16#81A5;
   // GBK_TO_UNICODE[203] := 16#4EF4;
   // GBK_TO_UNICODE[204] := 16#81A6;
   // GBK_TO_UNICODE[205] := 16#4EF8;
   // GBK_TO_UNICODE[206] := 16#81A7;
   // GBK_TO_UNICODE[207] := 16#4EF9;
   // GBK_TO_UNICODE[208] := 16#81A8;
   // GBK_TO_UNICODE[209] := 16#4EFA;
   // GBK_TO_UNICODE[210] := 16#81A9;
   // GBK_TO_UNICODE[211] := 16#4EFC;
   // GBK_TO_UNICODE[212] := 16#81AA;
   // GBK_TO_UNICODE[213] := 16#4EFE;
   // GBK_TO_UNICODE[214] := 16#81AB;
   // GBK_TO_UNICODE[215] := 16#4F00;
   // GBK_TO_UNICODE[216] := 16#81AC;
   // GBK_TO_UNICODE[217] := 16#4F02;
   // GBK_TO_UNICODE[218] := 16#81AD;
   // GBK_TO_UNICODE[219] := 16#4F03;
   // GBK_TO_UNICODE[220] := 16#81AE;
   // GBK_TO_UNICODE[221] := 16#4F04;
   // GBK_TO_UNICODE[222] := 16#81AF;
   // GBK_TO_UNICODE[223] := 16#4F05;
   // GBK_TO_UNICODE[224] := 16#81B0;
   // GBK_TO_UNICODE[225] := 16#4F06;
   // GBK_TO_UNICODE[226] := 16#81B1;
   // GBK_TO_UNICODE[227] := 16#4F07;
   // GBK_TO_UNICODE[228] := 16#81B2;
   // GBK_TO_UNICODE[229] := 16#4F08;
   // GBK_TO_UNICODE[230] := 16#81B3;
   // GBK_TO_UNICODE[231] := 16#4F0B;
   // GBK_TO_UNICODE[232] := 16#81B4;
   // GBK_TO_UNICODE[233] := 16#4F0C;
   // GBK_TO_UNICODE[234] := 16#81B5;
   // GBK_TO_UNICODE[235] := 16#4F12;
   // GBK_TO_UNICODE[236] := 16#81B6;
   // GBK_TO_UNICODE[237] := 16#4F13;
   // GBK_TO_UNICODE[238] := 16#81B7;
   // GBK_TO_UNICODE[239] := 16#4F14;
   // GBK_TO_UNICODE[240] := 16#81B8;
   // GBK_TO_UNICODE[241] := 16#4F15;
   // GBK_TO_UNICODE[242] := 16#81B9;
   // GBK_TO_UNICODE[243] := 16#4F16;
   // GBK_TO_UNICODE[244] := 16#81BA;
   // GBK_TO_UNICODE[245] := 16#4F1C;
   // GBK_TO_UNICODE[246] := 16#81BB;
   // GBK_TO_UNICODE[247] := 16#4F1D;
   // GBK_TO_UNICODE[248] := 16#81BC;
   // GBK_TO_UNICODE[249] := 16#4F21;
   // GBK_TO_UNICODE[250] := 16#81BD;
   // GBK_TO_UNICODE[251] := 16#4F23;
   // GBK_TO_UNICODE[252] := 16#81BE;
   // GBK_TO_UNICODE[253] := 16#4F28;
   // GBK_TO_UNICODE[254] := 16#81BF;
   // GBK_TO_UNICODE[255] := 16#4F29;
   // GBK_TO_UNICODE[256] := 16#81C0;
   // GBK_TO_UNICODE[257] := 16#4F2C;
   // GBK_TO_UNICODE[258] := 16#81C1;
   // GBK_TO_UNICODE[259] := 16#4F2D;
   // GBK_TO_UNICODE[260] := 16#81C2;
   // GBK_TO_UNICODE[261] := 16#4F2E;
   // GBK_TO_UNICODE[262] := 16#81C3;
   // GBK_TO_UNICODE[263] := 16#4F31;
   // GBK_TO_UNICODE[264] := 16#81C4;
   // GBK_TO_UNICODE[265] := 16#4F33;
   // GBK_TO_UNICODE[266] := 16#81C5;
   // GBK_TO_UNICODE[267] := 16#4F35;
   // GBK_TO_UNICODE[268] := 16#81C6;
   // GBK_TO_UNICODE[269] := 16#4F37;
   // GBK_TO_UNICODE[270] := 16#81C7;
   // GBK_TO_UNICODE[271] := 16#4F39;
   // GBK_TO_UNICODE[272] := 16#81C8;
   // GBK_TO_UNICODE[273] := 16#4F3B;
   // GBK_TO_UNICODE[274] := 16#81C9;
   // GBK_TO_UNICODE[275] := 16#4F3E;
   // GBK_TO_UNICODE[276] := 16#81CA;
   // GBK_TO_UNICODE[277] := 16#4F3F;
   // GBK_TO_UNICODE[278] := 16#81CB;
   // GBK_TO_UNICODE[279] := 16#4F40;
   // GBK_TO_UNICODE[280] := 16#81CC;
   // GBK_TO_UNICODE[281] := 16#4F41;
   // GBK_TO_UNICODE[282] := 16#81CD;
   // GBK_TO_UNICODE[283] := 16#4F42;
   // GBK_TO_UNICODE[284] := 16#81CE;
   // GBK_TO_UNICODE[285] := 16#4F44;
   // GBK_TO_UNICODE[286] := 16#81CF;
   // GBK_TO_UNICODE[287] := 16#4F45;
   // GBK_TO_UNICODE[288] := 16#81D0;
   // GBK_TO_UNICODE[289] := 16#4F47;
   // GBK_TO_UNICODE[290] := 16#81D1;
   // GBK_TO_UNICODE[291] := 16#4F48;
   // GBK_TO_UNICODE[292] := 16#81D2;
   // GBK_TO_UNICODE[293] := 16#4F49;
   // GBK_TO_UNICODE[294] := 16#81D3;
   // GBK_TO_UNICODE[295] := 16#4F4A;
   // GBK_TO_UNICODE[296] := 16#81D4;
   // GBK_TO_UNICODE[297] := 16#4F4B;
   // GBK_TO_UNICODE[298] := 16#81D5;
   // GBK_TO_UNICODE[299] := 16#4F4C;
   // GBK_TO_UNICODE[300] := 16#81D6;
   // GBK_TO_UNICODE[301] := 16#4F52;
   // GBK_TO_UNICODE[302] := 16#81D7;
   // GBK_TO_UNICODE[303] := 16#4F54;
   // GBK_TO_UNICODE[304] := 16#81D8;
   // GBK_TO_UNICODE[305] := 16#4F56;
   // GBK_TO_UNICODE[306] := 16#81D9;
   // GBK_TO_UNICODE[307] := 16#4F61;
   // GBK_TO_UNICODE[308] := 16#81DA;
   // GBK_TO_UNICODE[309] := 16#4F62;
   // GBK_TO_UNICODE[310] := 16#81DB;
   // GBK_TO_UNICODE[311] := 16#4F66;
   // GBK_TO_UNICODE[312] := 16#81DC;
   // GBK_TO_UNICODE[313] := 16#4F68;
   // GBK_TO_UNICODE[314] := 16#81DD;
   // GBK_TO_UNICODE[315] := 16#4F6A;
   // GBK_TO_UNICODE[316] := 16#81DE;
   // GBK_TO_UNICODE[317] := 16#4F6B;
   // GBK_TO_UNICODE[318] := 16#81DF;
   // GBK_TO_UNICODE[319] := 16#4F6D;
   // GBK_TO_UNICODE[320] := 16#81E0;
   // GBK_TO_UNICODE[321] := 16#4F6E;
   // GBK_TO_UNICODE[322] := 16#81E1;
   // GBK_TO_UNICODE[323] := 16#4F71;
   // GBK_TO_UNICODE[324] := 16#81E2;
   // GBK_TO_UNICODE[325] := 16#4F72;
   // GBK_TO_UNICODE[326] := 16#81E3;
   // GBK_TO_UNICODE[327] := 16#4F75;
   // GBK_TO_UNICODE[328] := 16#81E4;
   // GBK_TO_UNICODE[329] := 16#4F77;
   // GBK_TO_UNICODE[330] := 16#81E5;
   // GBK_TO_UNICODE[331] := 16#4F78;
   // GBK_TO_UNICODE[332] := 16#81E6;
   // GBK_TO_UNICODE[333] := 16#4F79;
   // GBK_TO_UNICODE[334] := 16#81E7;
   // GBK_TO_UNICODE[335] := 16#4F7A;
   // GBK_TO_UNICODE[336] := 16#81E8;
   // GBK_TO_UNICODE[337] := 16#4F7D;
   // GBK_TO_UNICODE[338] := 16#81E9;
   // GBK_TO_UNICODE[339] := 16#4F80;
   // GBK_TO_UNICODE[340] := 16#81EA;
   // GBK_TO_UNICODE[341] := 16#4F81;
   // GBK_TO_UNICODE[342] := 16#81EB;
   // GBK_TO_UNICODE[343] := 16#4F82;
   // GBK_TO_UNICODE[344] := 16#81EC;
   // GBK_TO_UNICODE[345] := 16#4F85;
   // GBK_TO_UNICODE[346] := 16#81ED;
   // GBK_TO_UNICODE[347] := 16#4F86;
   // GBK_TO_UNICODE[348] := 16#81EE;
   // GBK_TO_UNICODE[349] := 16#4F87;
   // GBK_TO_UNICODE[350] := 16#81EF;
   // GBK_TO_UNICODE[351] := 16#4F8A;
   // GBK_TO_UNICODE[352] := 16#81F0;
   // GBK_TO_UNICODE[353] := 16#4F8C;
   // GBK_TO_UNICODE[354] := 16#81F1;
   // GBK_TO_UNICODE[355] := 16#4F8E;
   // GBK_TO_UNICODE[356] := 16#81F2;
   // GBK_TO_UNICODE[357] := 16#4F90;
   // GBK_TO_UNICODE[358] := 16#81F3;
   // GBK_TO_UNICODE[359] := 16#4F92;
   // GBK_TO_UNICODE[360] := 16#81F4;
   // GBK_TO_UNICODE[361] := 16#4F93;
   // GBK_TO_UNICODE[362] := 16#81F5;
   // GBK_TO_UNICODE[363] := 16#4F95;
   // GBK_TO_UNICODE[364] := 16#81F6;
   // GBK_TO_UNICODE[365] := 16#4F96;
   // GBK_TO_UNICODE[366] := 16#81F7;
   // GBK_TO_UNICODE[367] := 16#4F98;
   // GBK_TO_UNICODE[368] := 16#81F8;
   // GBK_TO_UNICODE[369] := 16#4F99;
   // GBK_TO_UNICODE[370] := 16#81F9;
   // GBK_TO_UNICODE[371] := 16#4F9A;
   // GBK_TO_UNICODE[372] := 16#81FA;
   // GBK_TO_UNICODE[373] := 16#4F9C;
   // GBK_TO_UNICODE[374] := 16#81FB;
   // GBK_TO_UNICODE[375] := 16#4F9E;
   // GBK_TO_UNICODE[376] := 16#81FC;
   // GBK_TO_UNICODE[377] := 16#4F9F;
   // GBK_TO_UNICODE[378] := 16#81FD;
   // GBK_TO_UNICODE[379] := 16#4FA1;
   // GBK_TO_UNICODE[380] := 16#81FE;
   // GBK_TO_UNICODE[381] := 16#4FA2;
   // GBK_TO_UNICODE[382] := 16#8240;
   // GBK_TO_UNICODE[383] := 16#4FA4;
   // GBK_TO_UNICODE[384] := 16#8241;
   // GBK_TO_UNICODE[385] := 16#4FAB;
   // GBK_TO_UNICODE[386] := 16#8242;
   // GBK_TO_UNICODE[387] := 16#4FAD;
   // GBK_TO_UNICODE[388] := 16#8243;
   // GBK_TO_UNICODE[389] := 16#4FB0;
   // GBK_TO_UNICODE[390] := 16#8244;
   // GBK_TO_UNICODE[391] := 16#4FB1;
   // GBK_TO_UNICODE[392] := 16#8245;
   // GBK_TO_UNICODE[393] := 16#4FB2;
   // GBK_TO_UNICODE[394] := 16#8246;
   // GBK_TO_UNICODE[395] := 16#4FB3;
   // GBK_TO_UNICODE[396] := 16#8247;
   // GBK_TO_UNICODE[397] := 16#4FB4;
   // GBK_TO_UNICODE[398] := 16#8248;
   // GBK_TO_UNICODE[399] := 16#4FB6;
   // GBK_TO_UNICODE[400] := 16#8249;
   // GBK_TO_UNICODE[401] := 16#4FB7;
   // GBK_TO_UNICODE[402] := 16#824A;
   // GBK_TO_UNICODE[403] := 16#4FB8;
   // GBK_TO_UNICODE[404] := 16#824B;
   // GBK_TO_UNICODE[405] := 16#4FB9;
   // GBK_TO_UNICODE[406] := 16#824C;
   // GBK_TO_UNICODE[407] := 16#4FBA;
   // GBK_TO_UNICODE[408] := 16#824D;
   // GBK_TO_UNICODE[409] := 16#4FBB;
   // GBK_TO_UNICODE[410] := 16#824E;
   // GBK_TO_UNICODE[411] := 16#4FBC;
   // GBK_TO_UNICODE[412] := 16#824F;
   // GBK_TO_UNICODE[413] := 16#4FBD;
   // GBK_TO_UNICODE[414] := 16#8250;
   // GBK_TO_UNICODE[415] := 16#4FBE;
   // GBK_TO_UNICODE[416] := 16#8251;
   // GBK_TO_UNICODE[417] := 16#4FC0;
   // GBK_TO_UNICODE[418] := 16#8252;
   // GBK_TO_UNICODE[419] := 16#4FC1;
   // GBK_TO_UNICODE[420] := 16#8253;
   // GBK_TO_UNICODE[421] := 16#4FC2;
   // GBK_TO_UNICODE[422] := 16#8254;
   // GBK_TO_UNICODE[423] := 16#4FC6;
   // GBK_TO_UNICODE[424] := 16#8255;
   // GBK_TO_UNICODE[425] := 16#4FC7;
   // GBK_TO_UNICODE[426] := 16#8256;
   // GBK_TO_UNICODE[427] := 16#4FC8;
   // GBK_TO_UNICODE[428] := 16#8257;
   // GBK_TO_UNICODE[429] := 16#4FC9;
   // GBK_TO_UNICODE[430] := 16#8258;
   // GBK_TO_UNICODE[431] := 16#4FCB;
   // GBK_TO_UNICODE[432] := 16#8259;
   // GBK_TO_UNICODE[433] := 16#4FCC;
   // GBK_TO_UNICODE[434] := 16#825A;
   // GBK_TO_UNICODE[435] := 16#4FCD;
   // GBK_TO_UNICODE[436] := 16#825B;
   // GBK_TO_UNICODE[437] := 16#4FD2;
   // GBK_TO_UNICODE[438] := 16#825C;
   // GBK_TO_UNICODE[439] := 16#4FD3;
   // GBK_TO_UNICODE[440] := 16#825D;
   // GBK_TO_UNICODE[441] := 16#4FD4;
   // GBK_TO_UNICODE[442] := 16#825E;
   // GBK_TO_UNICODE[443] := 16#4FD5;
   // GBK_TO_UNICODE[444] := 16#825F;
   // GBK_TO_UNICODE[445] := 16#4FD6;
   // GBK_TO_UNICODE[446] := 16#8260;
   // GBK_TO_UNICODE[447] := 16#4FD9;
   // GBK_TO_UNICODE[448] := 16#8261;
   // GBK_TO_UNICODE[449] := 16#4FDB;
   // GBK_TO_UNICODE[450] := 16#8262;
   // GBK_TO_UNICODE[451] := 16#4FE0;
   // GBK_TO_UNICODE[452] := 16#8263;
   // GBK_TO_UNICODE[453] := 16#4FE2;
   // GBK_TO_UNICODE[454] := 16#8264;
   // GBK_TO_UNICODE[455] := 16#4FE4;
   // GBK_TO_UNICODE[456] := 16#8265;
   // GBK_TO_UNICODE[457] := 16#4FE5;
   // GBK_TO_UNICODE[458] := 16#8266;
   // GBK_TO_UNICODE[459] := 16#4FE7;
   // GBK_TO_UNICODE[460] := 16#8267;
   // GBK_TO_UNICODE[461] := 16#4FEB;
   // GBK_TO_UNICODE[462] := 16#8268;
   // GBK_TO_UNICODE[463] := 16#4FEC;
   // GBK_TO_UNICODE[464] := 16#8269;
   // GBK_TO_UNICODE[465] := 16#4FF0;
   // GBK_TO_UNICODE[466] := 16#826A;
   // GBK_TO_UNICODE[467] := 16#4FF2;
   // GBK_TO_UNICODE[468] := 16#826B;
   // GBK_TO_UNICODE[469] := 16#4FF4;
   // GBK_TO_UNICODE[470] := 16#826C;
   // GBK_TO_UNICODE[471] := 16#4FF5;
   // GBK_TO_UNICODE[472] := 16#826D;
   // GBK_TO_UNICODE[473] := 16#4FF6;
   // GBK_TO_UNICODE[474] := 16#826E;
   // GBK_TO_UNICODE[475] := 16#4FF7;
   // GBK_TO_UNICODE[476] := 16#826F;
   // GBK_TO_UNICODE[477] := 16#4FF9;
   // GBK_TO_UNICODE[478] := 16#8270;
   // GBK_TO_UNICODE[479] := 16#4FFB;
   // GBK_TO_UNICODE[480] := 16#8271;
   // GBK_TO_UNICODE[481] := 16#4FFC;
   // GBK_TO_UNICODE[482] := 16#8272;
   // GBK_TO_UNICODE[483] := 16#4FFD;
   // GBK_TO_UNICODE[484] := 16#8273;
   // GBK_TO_UNICODE[485] := 16#4FFF;
   // GBK_TO_UNICODE[486] := 16#8274;
   // GBK_TO_UNICODE[487] := 16#5000;
   // GBK_TO_UNICODE[488] := 16#8275;
   // GBK_TO_UNICODE[489] := 16#5001;
   // GBK_TO_UNICODE[490] := 16#8276;
   // GBK_TO_UNICODE[491] := 16#5002;
   // GBK_TO_UNICODE[492] := 16#8277;
   // GBK_TO_UNICODE[493] := 16#5003;
   // GBK_TO_UNICODE[494] := 16#8278;
   // GBK_TO_UNICODE[495] := 16#5004;
   // GBK_TO_UNICODE[496] := 16#8279;
   // GBK_TO_UNICODE[497] := 16#5005;
   // GBK_TO_UNICODE[498] := 16#827A;
   // GBK_TO_UNICODE[499] := 16#5006;
   // GBK_TO_UNICODE[500] := 16#827B;
   // GBK_TO_UNICODE[501] := 16#5007;
   // GBK_TO_UNICODE[502] := 16#827C;
   // GBK_TO_UNICODE[503] := 16#5008;
   // GBK_TO_UNICODE[504] := 16#827D;
   // GBK_TO_UNICODE[505] := 16#5009;
   // GBK_TO_UNICODE[506] := 16#827E;
   // GBK_TO_UNICODE[507] := 16#500A;
   // GBK_TO_UNICODE[508] := 16#8280;
   // GBK_TO_UNICODE[509] := 16#500B;
   // GBK_TO_UNICODE[510] := 16#8281;
   // GBK_TO_UNICODE[511] := 16#500E;
   // GBK_TO_UNICODE[512] := 16#8282;
   // GBK_TO_UNICODE[513] := 16#5010;
   // GBK_TO_UNICODE[514] := 16#8283;
   // GBK_TO_UNICODE[515] := 16#5011;
   // GBK_TO_UNICODE[516] := 16#8284;
   // GBK_TO_UNICODE[517] := 16#5013;
   // GBK_TO_UNICODE[518] := 16#8285;
   // GBK_TO_UNICODE[519] := 16#5015;
   // GBK_TO_UNICODE[520] := 16#8286;
   // GBK_TO_UNICODE[521] := 16#5016;
   // GBK_TO_UNICODE[522] := 16#8287;
   // GBK_TO_UNICODE[523] := 16#5017;
   // GBK_TO_UNICODE[524] := 16#8288;
   // GBK_TO_UNICODE[525] := 16#501B;
   // GBK_TO_UNICODE[526] := 16#8289;
   // GBK_TO_UNICODE[527] := 16#501D;
   // GBK_TO_UNICODE[528] := 16#828A;
   // GBK_TO_UNICODE[529] := 16#501E;
   // GBK_TO_UNICODE[530] := 16#828B;
   // GBK_TO_UNICODE[531] := 16#5020;
   // GBK_TO_UNICODE[532] := 16#828C;
   // GBK_TO_UNICODE[533] := 16#5022;
   // GBK_TO_UNICODE[534] := 16#828D;
   // GBK_TO_UNICODE[535] := 16#5023;
   // GBK_TO_UNICODE[536] := 16#828E;
   // GBK_TO_UNICODE[537] := 16#5024;
   // GBK_TO_UNICODE[538] := 16#828F;
   // GBK_TO_UNICODE[539] := 16#5027;
   // GBK_TO_UNICODE[540] := 16#8290;
   // GBK_TO_UNICODE[541] := 16#502B;
   // GBK_TO_UNICODE[542] := 16#8291;
   // GBK_TO_UNICODE[543] := 16#502F;
   // GBK_TO_UNICODE[544] := 16#8292;
   // GBK_TO_UNICODE[545] := 16#5030;
   // GBK_TO_UNICODE[546] := 16#8293;
   // GBK_TO_UNICODE[547] := 16#5031;
   // GBK_TO_UNICODE[548] := 16#8294;
   // GBK_TO_UNICODE[549] := 16#5032;
   // GBK_TO_UNICODE[550] := 16#8295;
   // GBK_TO_UNICODE[551] := 16#5033;
   // GBK_TO_UNICODE[552] := 16#8296;
   // GBK_TO_UNICODE[553] := 16#5034;
   // GBK_TO_UNICODE[554] := 16#8297;
   // GBK_TO_UNICODE[555] := 16#5035;
   // GBK_TO_UNICODE[556] := 16#8298;
   // GBK_TO_UNICODE[557] := 16#5036;
   // GBK_TO_UNICODE[558] := 16#8299;
   // GBK_TO_UNICODE[559] := 16#5037;
   // GBK_TO_UNICODE[560] := 16#829A;
   // GBK_TO_UNICODE[561] := 16#5038;
   // GBK_TO_UNICODE[562] := 16#829B;
   // GBK_TO_UNICODE[563] := 16#5039;
   // GBK_TO_UNICODE[564] := 16#829C;
   // GBK_TO_UNICODE[565] := 16#503B;
   // GBK_TO_UNICODE[566] := 16#829D;
   // GBK_TO_UNICODE[567] := 16#503D;
   // GBK_TO_UNICODE[568] := 16#829E;
   // GBK_TO_UNICODE[569] := 16#503F;
   // GBK_TO_UNICODE[570] := 16#829F;
   // GBK_TO_UNICODE[571] := 16#5040;
   // GBK_TO_UNICODE[572] := 16#82A0;
   // GBK_TO_UNICODE[573] := 16#5041;
   // GBK_TO_UNICODE[574] := 16#82A1;
   // GBK_TO_UNICODE[575] := 16#5042;
   // GBK_TO_UNICODE[576] := 16#82A2;
   // GBK_TO_UNICODE[577] := 16#5044;
   // GBK_TO_UNICODE[578] := 16#82A3;
   // GBK_TO_UNICODE[579] := 16#5045;
   // GBK_TO_UNICODE[580] := 16#82A4;
   // GBK_TO_UNICODE[581] := 16#5046;
   // GBK_TO_UNICODE[582] := 16#82A5;
   // GBK_TO_UNICODE[583] := 16#5049;
   // GBK_TO_UNICODE[584] := 16#82A6;
   // GBK_TO_UNICODE[585] := 16#504A;
   // GBK_TO_UNICODE[586] := 16#82A7;
   // GBK_TO_UNICODE[587] := 16#504B;
   // GBK_TO_UNICODE[588] := 16#82A8;
   // GBK_TO_UNICODE[589] := 16#504D;
   // GBK_TO_UNICODE[590] := 16#82A9;
   // GBK_TO_UNICODE[591] := 16#5050;
   // GBK_TO_UNICODE[592] := 16#82AA;
   // GBK_TO_UNICODE[593] := 16#5051;
   // GBK_TO_UNICODE[594] := 16#82AB;
   // GBK_TO_UNICODE[595] := 16#5052;
   // GBK_TO_UNICODE[596] := 16#82AC;
   // GBK_TO_UNICODE[597] := 16#5053;
   // GBK_TO_UNICODE[598] := 16#82AD;
   // GBK_TO_UNICODE[599] := 16#5054;
   // GBK_TO_UNICODE[600] := 16#82AE;
   // GBK_TO_UNICODE[601] := 16#5056;
   // GBK_TO_UNICODE[602] := 16#82AF;
   // GBK_TO_UNICODE[603] := 16#5057;
   // GBK_TO_UNICODE[604] := 16#82B0;
   // GBK_TO_UNICODE[605] := 16#5058;
   // GBK_TO_UNICODE[606] := 16#82B1;
   // GBK_TO_UNICODE[607] := 16#5059;
   // GBK_TO_UNICODE[608] := 16#82B2;
   // GBK_TO_UNICODE[609] := 16#505B;
   // GBK_TO_UNICODE[610] := 16#82B3;
   // GBK_TO_UNICODE[611] := 16#505D;
   // GBK_TO_UNICODE[612] := 16#82B4;
   // GBK_TO_UNICODE[613] := 16#505E;
   // GBK_TO_UNICODE[614] := 16#82B5;
   // GBK_TO_UNICODE[615] := 16#505F;
   // GBK_TO_UNICODE[616] := 16#82B6;
   // GBK_TO_UNICODE[617] := 16#5060;
   // GBK_TO_UNICODE[618] := 16#82B7;
   // GBK_TO_UNICODE[619] := 16#5061;
   // GBK_TO_UNICODE[620] := 16#82B8;
   // GBK_TO_UNICODE[621] := 16#5062;
   // GBK_TO_UNICODE[622] := 16#82B9;
   // GBK_TO_UNICODE[623] := 16#5063;
   // GBK_TO_UNICODE[624] := 16#82BA;
   // GBK_TO_UNICODE[625] := 16#5064;
   // GBK_TO_UNICODE[626] := 16#82BB;
   // GBK_TO_UNICODE[627] := 16#5066;
   // GBK_TO_UNICODE[628] := 16#82BC;
   // GBK_TO_UNICODE[629] := 16#5067;
   // GBK_TO_UNICODE[630] := 16#82BD;
   // GBK_TO_UNICODE[631] := 16#5068;
   // GBK_TO_UNICODE[632] := 16#82BE;
   // GBK_TO_UNICODE[633] := 16#5069;
   // GBK_TO_UNICODE[634] := 16#82BF;
   // GBK_TO_UNICODE[635] := 16#506A;
   // GBK_TO_UNICODE[636] := 16#82C0;
   // GBK_TO_UNICODE[637] := 16#506B;
   // GBK_TO_UNICODE[638] := 16#82C1;
   // GBK_TO_UNICODE[639] := 16#506D;
   // GBK_TO_UNICODE[640] := 16#82C2;
   // GBK_TO_UNICODE[641] := 16#506E;
   // GBK_TO_UNICODE[642] := 16#82C3;
   // GBK_TO_UNICODE[643] := 16#506F;
   // GBK_TO_UNICODE[644] := 16#82C4;
   // GBK_TO_UNICODE[645] := 16#5070;
   // GBK_TO_UNICODE[646] := 16#82C5;
   // GBK_TO_UNICODE[647] := 16#5071;
   // GBK_TO_UNICODE[648] := 16#82C6;
   // GBK_TO_UNICODE[649] := 16#5072;
   // GBK_TO_UNICODE[650] := 16#82C7;
   // GBK_TO_UNICODE[651] := 16#5073;
   // GBK_TO_UNICODE[652] := 16#82C8;
   // GBK_TO_UNICODE[653] := 16#5074;
   // GBK_TO_UNICODE[654] := 16#82C9;
   // GBK_TO_UNICODE[655] := 16#5075;
   // GBK_TO_UNICODE[656] := 16#82CA;
   // GBK_TO_UNICODE[657] := 16#5078;
   // GBK_TO_UNICODE[658] := 16#82CB;
   // GBK_TO_UNICODE[659] := 16#5079;
   // GBK_TO_UNICODE[660] := 16#82CC;
   // GBK_TO_UNICODE[661] := 16#507A;
   // GBK_TO_UNICODE[662] := 16#82CD;
   // GBK_TO_UNICODE[663] := 16#507C;
   // GBK_TO_UNICODE[664] := 16#82CE;
   // GBK_TO_UNICODE[665] := 16#507D;
   // GBK_TO_UNICODE[666] := 16#82CF;
   // GBK_TO_UNICODE[667] := 16#5081;
   // GBK_TO_UNICODE[668] := 16#82D0;
   // GBK_TO_UNICODE[669] := 16#5082;
   // GBK_TO_UNICODE[670] := 16#82D1;
   // GBK_TO_UNICODE[671] := 16#5083;
   // GBK_TO_UNICODE[672] := 16#82D2;
   // GBK_TO_UNICODE[673] := 16#5084;
   // GBK_TO_UNICODE[674] := 16#82D3;
   // GBK_TO_UNICODE[675] := 16#5086;
   // GBK_TO_UNICODE[676] := 16#82D4;
   // GBK_TO_UNICODE[677] := 16#5087;
   // GBK_TO_UNICODE[678] := 16#82D5;
   // GBK_TO_UNICODE[679] := 16#5089;
   // GBK_TO_UNICODE[680] := 16#82D6;
   // GBK_TO_UNICODE[681] := 16#508A;
   // GBK_TO_UNICODE[682] := 16#82D7;
   // GBK_TO_UNICODE[683] := 16#508B;
   // GBK_TO_UNICODE[684] := 16#82D8;
   // GBK_TO_UNICODE[685] := 16#508C;
   // GBK_TO_UNICODE[686] := 16#82D9;
   // GBK_TO_UNICODE[687] := 16#508E;
   // GBK_TO_UNICODE[688] := 16#82DA;
   // GBK_TO_UNICODE[689] := 16#508F;
   // GBK_TO_UNICODE[690] := 16#82DB;
   // GBK_TO_UNICODE[691] := 16#5090;
   // GBK_TO_UNICODE[692] := 16#82DC;
   // GBK_TO_UNICODE[693] := 16#5091;
   // GBK_TO_UNICODE[694] := 16#82DD;
   // GBK_TO_UNICODE[695] := 16#5092;
   // GBK_TO_UNICODE[696] := 16#82DE;
   // GBK_TO_UNICODE[697] := 16#5093;
   // GBK_TO_UNICODE[698] := 16#82DF;
   // GBK_TO_UNICODE[699] := 16#5094;
   // GBK_TO_UNICODE[700] := 16#82E0;
   // GBK_TO_UNICODE[701] := 16#5095;
   // GBK_TO_UNICODE[702] := 16#82E1;
   // GBK_TO_UNICODE[703] := 16#5096;
   // GBK_TO_UNICODE[704] := 16#82E2;
   // GBK_TO_UNICODE[705] := 16#5097;
   // GBK_TO_UNICODE[706] := 16#82E3;
   // GBK_TO_UNICODE[707] := 16#5098;
   // GBK_TO_UNICODE[708] := 16#82E4;
   // GBK_TO_UNICODE[709] := 16#5099;
   // GBK_TO_UNICODE[710] := 16#82E5;
   // GBK_TO_UNICODE[711] := 16#509A;
   // GBK_TO_UNICODE[712] := 16#82E6;
   // GBK_TO_UNICODE[713] := 16#509B;
   // GBK_TO_UNICODE[714] := 16#82E7;
   // GBK_TO_UNICODE[715] := 16#509C;
   // GBK_TO_UNICODE[716] := 16#82E8;
   // GBK_TO_UNICODE[717] := 16#509D;
   // GBK_TO_UNICODE[718] := 16#82E9;
   // GBK_TO_UNICODE[719] := 16#509E;
   // GBK_TO_UNICODE[720] := 16#82EA;
   // GBK_TO_UNICODE[721] := 16#509F;
   // GBK_TO_UNICODE[722] := 16#82EB;
   // GBK_TO_UNICODE[723] := 16#50A0;
   // GBK_TO_UNICODE[724] := 16#82EC;
   // GBK_TO_UNICODE[725] := 16#50A1;
   // GBK_TO_UNICODE[726] := 16#82ED;
   // GBK_TO_UNICODE[727] := 16#50A2;
   // GBK_TO_UNICODE[728] := 16#82EE;
   // GBK_TO_UNICODE[729] := 16#50A4;
   // GBK_TO_UNICODE[730] := 16#82EF;
   // GBK_TO_UNICODE[731] := 16#50A6;
   // GBK_TO_UNICODE[732] := 16#82F0;
   // GBK_TO_UNICODE[733] := 16#50AA;
   // GBK_TO_UNICODE[734] := 16#82F1;
   // GBK_TO_UNICODE[735] := 16#50AB;
   // GBK_TO_UNICODE[736] := 16#82F2;
   // GBK_TO_UNICODE[737] := 16#50AD;
   // GBK_TO_UNICODE[738] := 16#82F3;
   // GBK_TO_UNICODE[739] := 16#50AE;
   // GBK_TO_UNICODE[740] := 16#82F4;
   // GBK_TO_UNICODE[741] := 16#50AF;
   // GBK_TO_UNICODE[742] := 16#82F5;
   // GBK_TO_UNICODE[743] := 16#50B0;
   // GBK_TO_UNICODE[744] := 16#82F6;
   // GBK_TO_UNICODE[745] := 16#50B1;
   // GBK_TO_UNICODE[746] := 16#82F7;
   // GBK_TO_UNICODE[747] := 16#50B3;
   // GBK_TO_UNICODE[748] := 16#82F8;
   // GBK_TO_UNICODE[749] := 16#50B4;
   // GBK_TO_UNICODE[750] := 16#82F9;
   // GBK_TO_UNICODE[751] := 16#50B5;
   // GBK_TO_UNICODE[752] := 16#82FA;
   // GBK_TO_UNICODE[753] := 16#50B6;
   // GBK_TO_UNICODE[754] := 16#82FB;
   // GBK_TO_UNICODE[755] := 16#50B7;
   // GBK_TO_UNICODE[756] := 16#82FC;
   // GBK_TO_UNICODE[757] := 16#50B8;
   // GBK_TO_UNICODE[758] := 16#82FD;
   // GBK_TO_UNICODE[759] := 16#50B9;
   // GBK_TO_UNICODE[760] := 16#82FE;
   // GBK_TO_UNICODE[761] := 16#50BC;
   // GBK_TO_UNICODE[762] := 16#8340;
   // GBK_TO_UNICODE[763] := 16#50BD;
   // GBK_TO_UNICODE[764] := 16#8341;
   // GBK_TO_UNICODE[765] := 16#50BE;
   // GBK_TO_UNICODE[766] := 16#8342;
   // GBK_TO_UNICODE[767] := 16#50BF;
   // GBK_TO_UNICODE[768] := 16#8343;
   // GBK_TO_UNICODE[769] := 16#50C0;
   // GBK_TO_UNICODE[770] := 16#8344;
   // GBK_TO_UNICODE[771] := 16#50C1;
   // GBK_TO_UNICODE[772] := 16#8345;
   // GBK_TO_UNICODE[773] := 16#50C2;
   // GBK_TO_UNICODE[774] := 16#8346;
   // GBK_TO_UNICODE[775] := 16#50C3;
   // GBK_TO_UNICODE[776] := 16#8347;
   // GBK_TO_UNICODE[777] := 16#50C4;
   // GBK_TO_UNICODE[778] := 16#8348;
   // GBK_TO_UNICODE[779] := 16#50C5;
   // GBK_TO_UNICODE[780] := 16#8349;
   // GBK_TO_UNICODE[781] := 16#50C6;
   // GBK_TO_UNICODE[782] := 16#834A;
   // GBK_TO_UNICODE[783] := 16#50C7;
   // GBK_TO_UNICODE[784] := 16#834B;
   // GBK_TO_UNICODE[785] := 16#50C8;
   // GBK_TO_UNICODE[786] := 16#834C;
   // GBK_TO_UNICODE[787] := 16#50C9;
   // GBK_TO_UNICODE[788] := 16#834D;
   // GBK_TO_UNICODE[789] := 16#50CA;
   // GBK_TO_UNICODE[790] := 16#834E;
   // GBK_TO_UNICODE[791] := 16#50CB;
   // GBK_TO_UNICODE[792] := 16#834F;
   // GBK_TO_UNICODE[793] := 16#50CC;
   // GBK_TO_UNICODE[794] := 16#8350;
   // GBK_TO_UNICODE[795] := 16#50CD;
   // GBK_TO_UNICODE[796] := 16#8351;
   // GBK_TO_UNICODE[797] := 16#50CE;
   // GBK_TO_UNICODE[798] := 16#8352;
   // GBK_TO_UNICODE[799] := 16#50D0;
   // GBK_TO_UNICODE[800] := 16#8353;
   // GBK_TO_UNICODE[801] := 16#50D1;
   // GBK_TO_UNICODE[802] := 16#8354;
   // GBK_TO_UNICODE[803] := 16#50D2;
   // GBK_TO_UNICODE[804] := 16#8355;
   // GBK_TO_UNICODE[805] := 16#50D3;
   // GBK_TO_UNICODE[806] := 16#8356;
   // GBK_TO_UNICODE[807] := 16#50D4;
   // GBK_TO_UNICODE[808] := 16#8357;
   // GBK_TO_UNICODE[809] := 16#50D5;
   // GBK_TO_UNICODE[810] := 16#8358;
   // GBK_TO_UNICODE[811] := 16#50D7;
   // GBK_TO_UNICODE[812] := 16#8359;
   // GBK_TO_UNICODE[813] := 16#50D8;
   // GBK_TO_UNICODE[814] := 16#835A;
   // GBK_TO_UNICODE[815] := 16#50D9;
   // GBK_TO_UNICODE[816] := 16#835B;
   // GBK_TO_UNICODE[817] := 16#50DB;
   // GBK_TO_UNICODE[818] := 16#835C;
   // GBK_TO_UNICODE[819] := 16#50DC;
   // GBK_TO_UNICODE[820] := 16#835D;
   // GBK_TO_UNICODE[821] := 16#50DD;
   // GBK_TO_UNICODE[822] := 16#835E;
   // GBK_TO_UNICODE[823] := 16#50DE;
   // GBK_TO_UNICODE[824] := 16#835F;
   // GBK_TO_UNICODE[825] := 16#50DF;
   // GBK_TO_UNICODE[826] := 16#8360;
   // GBK_TO_UNICODE[827] := 16#50E0;
   // GBK_TO_UNICODE[828] := 16#8361;
   // GBK_TO_UNICODE[829] := 16#50E1;
   // GBK_TO_UNICODE[830] := 16#8362;
   // GBK_TO_UNICODE[831] := 16#50E2;
   // GBK_TO_UNICODE[832] := 16#8363;
   // GBK_TO_UNICODE[833] := 16#50E3;
   // GBK_TO_UNICODE[834] := 16#8364;
   // GBK_TO_UNICODE[835] := 16#50E4;
   // GBK_TO_UNICODE[836] := 16#8365;
   // GBK_TO_UNICODE[837] := 16#50E5;
   // GBK_TO_UNICODE[838] := 16#8366;
   // GBK_TO_UNICODE[839] := 16#50E8;
   // GBK_TO_UNICODE[840] := 16#8367;
   // GBK_TO_UNICODE[841] := 16#50E9;
   // GBK_TO_UNICODE[842] := 16#8368;
   // GBK_TO_UNICODE[843] := 16#50EA;
   // GBK_TO_UNICODE[844] := 16#8369;
   // GBK_TO_UNICODE[845] := 16#50EB;
   // GBK_TO_UNICODE[846] := 16#836A;
   // GBK_TO_UNICODE[847] := 16#50EF;
   // GBK_TO_UNICODE[848] := 16#836B;
   // GBK_TO_UNICODE[849] := 16#50F0;
   // GBK_TO_UNICODE[850] := 16#836C;
   // GBK_TO_UNICODE[851] := 16#50F1;
   // GBK_TO_UNICODE[852] := 16#836D;
   // GBK_TO_UNICODE[853] := 16#50F2;
   // GBK_TO_UNICODE[854] := 16#836E;
   // GBK_TO_UNICODE[855] := 16#50F4;
   // GBK_TO_UNICODE[856] := 16#836F;
   // GBK_TO_UNICODE[857] := 16#50F6;
   // GBK_TO_UNICODE[858] := 16#8370;
   // GBK_TO_UNICODE[859] := 16#50F7;
   // GBK_TO_UNICODE[860] := 16#8371;
   // GBK_TO_UNICODE[861] := 16#50F8;
   // GBK_TO_UNICODE[862] := 16#8372;
   // GBK_TO_UNICODE[863] := 16#50F9;
   // GBK_TO_UNICODE[864] := 16#8373;
   // GBK_TO_UNICODE[865] := 16#50FA;
   // GBK_TO_UNICODE[866] := 16#8374;
   // GBK_TO_UNICODE[867] := 16#50FC;
   // GBK_TO_UNICODE[868] := 16#8375;
   // GBK_TO_UNICODE[869] := 16#50FD;
   // GBK_TO_UNICODE[870] := 16#8376;
   // GBK_TO_UNICODE[871] := 16#50FE;
   // GBK_TO_UNICODE[872] := 16#8377;
   // GBK_TO_UNICODE[873] := 16#50FF;
   // GBK_TO_UNICODE[874] := 16#8378;
   // GBK_TO_UNICODE[875] := 16#5100;
   // GBK_TO_UNICODE[876] := 16#8379;
   // GBK_TO_UNICODE[877] := 16#5101;
   // GBK_TO_UNICODE[878] := 16#837A;
   // GBK_TO_UNICODE[879] := 16#5102;
   // GBK_TO_UNICODE[880] := 16#837B;
   // GBK_TO_UNICODE[881] := 16#5103;
   // GBK_TO_UNICODE[882] := 16#837C;
   // GBK_TO_UNICODE[883] := 16#5104;
   // GBK_TO_UNICODE[884] := 16#837D;
   // GBK_TO_UNICODE[885] := 16#5105;
   // GBK_TO_UNICODE[886] := 16#837E;
   // GBK_TO_UNICODE[887] := 16#5108;
   // GBK_TO_UNICODE[888] := 16#8380;
   // GBK_TO_UNICODE[889] := 16#5109;
   // GBK_TO_UNICODE[890] := 16#8381;
   // GBK_TO_UNICODE[891] := 16#510A;
   // GBK_TO_UNICODE[892] := 16#8382;
   // GBK_TO_UNICODE[893] := 16#510C;
   // GBK_TO_UNICODE[894] := 16#8383;
   // GBK_TO_UNICODE[895] := 16#510D;
   // GBK_TO_UNICODE[896] := 16#8384;
   // GBK_TO_UNICODE[897] := 16#510E;
   // GBK_TO_UNICODE[898] := 16#8385;
   // GBK_TO_UNICODE[899] := 16#510F;
   // GBK_TO_UNICODE[900] := 16#8386;
   // GBK_TO_UNICODE[901] := 16#5110;
   // GBK_TO_UNICODE[902] := 16#8387;
   // GBK_TO_UNICODE[903] := 16#5111;
   // GBK_TO_UNICODE[904] := 16#8388;
   // GBK_TO_UNICODE[905] := 16#5113;
   // GBK_TO_UNICODE[906] := 16#8389;
   // GBK_TO_UNICODE[907] := 16#5114;
   // GBK_TO_UNICODE[908] := 16#838A;
   // GBK_TO_UNICODE[909] := 16#5115;
   // GBK_TO_UNICODE[910] := 16#838B;
   // GBK_TO_UNICODE[911] := 16#5116;
   // GBK_TO_UNICODE[912] := 16#838C;
   // GBK_TO_UNICODE[913] := 16#5117;
   // GBK_TO_UNICODE[914] := 16#838D;
   // GBK_TO_UNICODE[915] := 16#5118;
   // GBK_TO_UNICODE[916] := 16#838E;
   // GBK_TO_UNICODE[917] := 16#5119;
   // GBK_TO_UNICODE[918] := 16#838F;
   // GBK_TO_UNICODE[919] := 16#511A;
   // GBK_TO_UNICODE[920] := 16#8390;
   // GBK_TO_UNICODE[921] := 16#511B;
   // GBK_TO_UNICODE[922] := 16#8391;
   // GBK_TO_UNICODE[923] := 16#511C;
   // GBK_TO_UNICODE[924] := 16#8392;
   // GBK_TO_UNICODE[925] := 16#511D;
   // GBK_TO_UNICODE[926] := 16#8393;
   // GBK_TO_UNICODE[927] := 16#511E;
   // GBK_TO_UNICODE[928] := 16#8394;
   // GBK_TO_UNICODE[929] := 16#511F;
   // GBK_TO_UNICODE[930] := 16#8395;
   // GBK_TO_UNICODE[931] := 16#5120;
   // GBK_TO_UNICODE[932] := 16#8396;
   // GBK_TO_UNICODE[933] := 16#5122;
   // GBK_TO_UNICODE[934] := 16#8397;
   // GBK_TO_UNICODE[935] := 16#5123;
   // GBK_TO_UNICODE[936] := 16#8398;
   // GBK_TO_UNICODE[937] := 16#5124;
   // GBK_TO_UNICODE[938] := 16#8399;
   // GBK_TO_UNICODE[939] := 16#5125;
   // GBK_TO_UNICODE[940] := 16#839A;
   // GBK_TO_UNICODE[941] := 16#5126;
   // GBK_TO_UNICODE[942] := 16#839B;
   // GBK_TO_UNICODE[943] := 16#5127;
   // GBK_TO_UNICODE[944] := 16#839C;
   // GBK_TO_UNICODE[945] := 16#5128;
   // GBK_TO_UNICODE[946] := 16#839D;
   // GBK_TO_UNICODE[947] := 16#5129;
   // GBK_TO_UNICODE[948] := 16#839E;
   // GBK_TO_UNICODE[949] := 16#512A;
   // GBK_TO_UNICODE[950] := 16#839F;
   // GBK_TO_UNICODE[951] := 16#512B;
   // GBK_TO_UNICODE[952] := 16#83A0;
   // GBK_TO_UNICODE[953] := 16#512C;
   // GBK_TO_UNICODE[954] := 16#83A1;
   // GBK_TO_UNICODE[955] := 16#512D;
   // GBK_TO_UNICODE[956] := 16#83A2;
   // GBK_TO_UNICODE[957] := 16#512E;
   // GBK_TO_UNICODE[958] := 16#83A3;
   // GBK_TO_UNICODE[959] := 16#512F;
   // GBK_TO_UNICODE[960] := 16#83A4;
   // GBK_TO_UNICODE[961] := 16#5130;
   // GBK_TO_UNICODE[962] := 16#83A5;
   // GBK_TO_UNICODE[963] := 16#5131;
   // GBK_TO_UNICODE[964] := 16#83A6;
   // GBK_TO_UNICODE[965] := 16#5132;
   // GBK_TO_UNICODE[966] := 16#83A7;
   // GBK_TO_UNICODE[967] := 16#5133;
   // GBK_TO_UNICODE[968] := 16#83A8;
   // GBK_TO_UNICODE[969] := 16#5134;
   // GBK_TO_UNICODE[970] := 16#83A9;
   // GBK_TO_UNICODE[971] := 16#5135;
   // GBK_TO_UNICODE[972] := 16#83AA;
   // GBK_TO_UNICODE[973] := 16#5136;
   // GBK_TO_UNICODE[974] := 16#83AB;
   // GBK_TO_UNICODE[975] := 16#5137;
   // GBK_TO_UNICODE[976] := 16#83AC;
   // GBK_TO_UNICODE[977] := 16#5138;
   // GBK_TO_UNICODE[978] := 16#83AD;
   // GBK_TO_UNICODE[979] := 16#5139;
   // GBK_TO_UNICODE[980] := 16#83AE;
   // GBK_TO_UNICODE[981] := 16#513A;
   // GBK_TO_UNICODE[982] := 16#83AF;
   // GBK_TO_UNICODE[983] := 16#513B;
   // GBK_TO_UNICODE[984] := 16#83B0;
   // GBK_TO_UNICODE[985] := 16#513C;
   // GBK_TO_UNICODE[986] := 16#83B1;
   // GBK_TO_UNICODE[987] := 16#513D;
   // GBK_TO_UNICODE[988] := 16#83B2;
   // GBK_TO_UNICODE[989] := 16#513E;
   // GBK_TO_UNICODE[990] := 16#83B3;
   // GBK_TO_UNICODE[991] := 16#5142;
   // GBK_TO_UNICODE[992] := 16#83B4;
   // GBK_TO_UNICODE[993] := 16#5147;
   // GBK_TO_UNICODE[994] := 16#83B5;
   // GBK_TO_UNICODE[995] := 16#514A;
   // GBK_TO_UNICODE[996] := 16#83B6;
   // GBK_TO_UNICODE[997] := 16#514C;
   // GBK_TO_UNICODE[998] := 16#83B7;
   // GBK_TO_UNICODE[999] := 16#514E;
   // GBK_TO_UNICODE[1000] := 16#83B8;
   // GBK_TO_UNICODE[1001] := 16#514F;
   // GBK_TO_UNICODE[1002] := 16#83B9;
   // GBK_TO_UNICODE[1003] := 16#5150;
   // GBK_TO_UNICODE[1004] := 16#83BA;
   // GBK_TO_UNICODE[1005] := 16#5152;
   // GBK_TO_UNICODE[1006] := 16#83BB;
   // GBK_TO_UNICODE[1007] := 16#5153;
   // GBK_TO_UNICODE[1008] := 16#83BC;
   // GBK_TO_UNICODE[1009] := 16#5157;
   // GBK_TO_UNICODE[1010] := 16#83BD;
   // GBK_TO_UNICODE[1011] := 16#5158;
   // GBK_TO_UNICODE[1012] := 16#83BE;
   // GBK_TO_UNICODE[1013] := 16#5159;
   // GBK_TO_UNICODE[1014] := 16#83BF;
   // GBK_TO_UNICODE[1015] := 16#515B;
   // GBK_TO_UNICODE[1016] := 16#83C0;
   // GBK_TO_UNICODE[1017] := 16#515D;
   // GBK_TO_UNICODE[1018] := 16#83C1;
   // GBK_TO_UNICODE[1019] := 16#515E;
   // GBK_TO_UNICODE[1020] := 16#83C2;
   // GBK_TO_UNICODE[1021] := 16#515F;
   // GBK_TO_UNICODE[1022] := 16#83C3;
   // GBK_TO_UNICODE[1023] := 16#5160;
   // GBK_TO_UNICODE[1024] := 16#83C4;
   // GBK_TO_UNICODE[1025] := 16#5161;
   // GBK_TO_UNICODE[1026] := 16#83C5;
   // GBK_TO_UNICODE[1027] := 16#5163;
   // GBK_TO_UNICODE[1028] := 16#83C6;
   // GBK_TO_UNICODE[1029] := 16#5164;
   // GBK_TO_UNICODE[1030] := 16#83C7;
   // GBK_TO_UNICODE[1031] := 16#5166;
   // GBK_TO_UNICODE[1032] := 16#83C8;
   // GBK_TO_UNICODE[1033] := 16#5167;
   // GBK_TO_UNICODE[1034] := 16#83C9;
   // GBK_TO_UNICODE[1035] := 16#5169;
   // GBK_TO_UNICODE[1036] := 16#83CA;
   // GBK_TO_UNICODE[1037] := 16#516A;
   // GBK_TO_UNICODE[1038] := 16#83CB;
   // GBK_TO_UNICODE[1039] := 16#516F;
   // GBK_TO_UNICODE[1040] := 16#83CC;
   // GBK_TO_UNICODE[1041] := 16#5172;
   // GBK_TO_UNICODE[1042] := 16#83CD;
   // GBK_TO_UNICODE[1043] := 16#517A;
   // GBK_TO_UNICODE[1044] := 16#83CE;
   // GBK_TO_UNICODE[1045] := 16#517E;
   // GBK_TO_UNICODE[1046] := 16#83CF;
   // GBK_TO_UNICODE[1047] := 16#517F;
   // GBK_TO_UNICODE[1048] := 16#83D0;
   // GBK_TO_UNICODE[1049] := 16#5183;
   // GBK_TO_UNICODE[1050] := 16#83D1;
   // GBK_TO_UNICODE[1051] := 16#5184;
   // GBK_TO_UNICODE[1052] := 16#83D2;
   // GBK_TO_UNICODE[1053] := 16#5186;
   // GBK_TO_UNICODE[1054] := 16#83D3;
   // GBK_TO_UNICODE[1055] := 16#5187;
   // GBK_TO_UNICODE[1056] := 16#83D4;
   // GBK_TO_UNICODE[1057] := 16#518A;
   // GBK_TO_UNICODE[1058] := 16#83D5;
   // GBK_TO_UNICODE[1059] := 16#518B;
   // GBK_TO_UNICODE[1060] := 16#83D6;
   // GBK_TO_UNICODE[1061] := 16#518E;
   // GBK_TO_UNICODE[1062] := 16#83D7;
   // GBK_TO_UNICODE[1063] := 16#518F;
   // GBK_TO_UNICODE[1064] := 16#83D8;
   // GBK_TO_UNICODE[1065] := 16#5190;
   // GBK_TO_UNICODE[1066] := 16#83D9;
   // GBK_TO_UNICODE[1067] := 16#5191;
   // GBK_TO_UNICODE[1068] := 16#83DA;
   // GBK_TO_UNICODE[1069] := 16#5193;
   // GBK_TO_UNICODE[1070] := 16#83DB;
   // GBK_TO_UNICODE[1071] := 16#5194;
   // GBK_TO_UNICODE[1072] := 16#83DC;
   // GBK_TO_UNICODE[1073] := 16#5198;
   // GBK_TO_UNICODE[1074] := 16#83DD;
   // GBK_TO_UNICODE[1075] := 16#519A;
   // GBK_TO_UNICODE[1076] := 16#83DE;
   // GBK_TO_UNICODE[1077] := 16#519D;
   // GBK_TO_UNICODE[1078] := 16#83DF;
   // GBK_TO_UNICODE[1079] := 16#519E;
   // GBK_TO_UNICODE[1080] := 16#83E0;
   // GBK_TO_UNICODE[1081] := 16#519F;
   // GBK_TO_UNICODE[1082] := 16#83E1;
   // GBK_TO_UNICODE[1083] := 16#51A1;
   // GBK_TO_UNICODE[1084] := 16#83E2;
   // GBK_TO_UNICODE[1085] := 16#51A3;
   // GBK_TO_UNICODE[1086] := 16#83E3;
   // GBK_TO_UNICODE[1087] := 16#51A6;
   // GBK_TO_UNICODE[1088] := 16#83E4;
   // GBK_TO_UNICODE[1089] := 16#51A7;
   // GBK_TO_UNICODE[1090] := 16#83E5;
   // GBK_TO_UNICODE[1091] := 16#51A8;
   // GBK_TO_UNICODE[1092] := 16#83E6;
   // GBK_TO_UNICODE[1093] := 16#51A9;
   // GBK_TO_UNICODE[1094] := 16#83E7;
   // GBK_TO_UNICODE[1095] := 16#51AA;
   // GBK_TO_UNICODE[1096] := 16#83E8;
   // GBK_TO_UNICODE[1097] := 16#51AD;
   // GBK_TO_UNICODE[1098] := 16#83E9;
   // GBK_TO_UNICODE[1099] := 16#51AE;
   // GBK_TO_UNICODE[1100] := 16#83EA;
   // GBK_TO_UNICODE[1101] := 16#51B4;
   // GBK_TO_UNICODE[1102] := 16#83EB;
   // GBK_TO_UNICODE[1103] := 16#51B8;
   // GBK_TO_UNICODE[1104] := 16#83EC;
   // GBK_TO_UNICODE[1105] := 16#51B9;
   // GBK_TO_UNICODE[1106] := 16#83ED;
   // GBK_TO_UNICODE[1107] := 16#51BA;
   // GBK_TO_UNICODE[1108] := 16#83EE;
   // GBK_TO_UNICODE[1109] := 16#51BE;
   // GBK_TO_UNICODE[1110] := 16#83EF;
   // GBK_TO_UNICODE[1111] := 16#51BF;
   // GBK_TO_UNICODE[1112] := 16#83F0;
   // GBK_TO_UNICODE[1113] := 16#51C1;
   // GBK_TO_UNICODE[1114] := 16#83F1;
   // GBK_TO_UNICODE[1115] := 16#51C2;
   // GBK_TO_UNICODE[1116] := 16#83F2;
   // GBK_TO_UNICODE[1117] := 16#51C3;
   // GBK_TO_UNICODE[1118] := 16#83F3;
   // GBK_TO_UNICODE[1119] := 16#51C5;
   // GBK_TO_UNICODE[1120] := 16#83F4;
   // GBK_TO_UNICODE[1121] := 16#51C8;
   // GBK_TO_UNICODE[1122] := 16#83F5;
   // GBK_TO_UNICODE[1123] := 16#51CA;
   // GBK_TO_UNICODE[1124] := 16#83F6;
   // GBK_TO_UNICODE[1125] := 16#51CD;
   // GBK_TO_UNICODE[1126] := 16#83F7;
   // GBK_TO_UNICODE[1127] := 16#51CE;
   // GBK_TO_UNICODE[1128] := 16#83F8;
   // GBK_TO_UNICODE[1129] := 16#51D0;
   // GBK_TO_UNICODE[1130] := 16#83F9;
   // GBK_TO_UNICODE[1131] := 16#51D2;
   // GBK_TO_UNICODE[1132] := 16#83FA;
   // GBK_TO_UNICODE[1133] := 16#51D3;
   // GBK_TO_UNICODE[1134] := 16#83FB;
   // GBK_TO_UNICODE[1135] := 16#51D4;
   // GBK_TO_UNICODE[1136] := 16#83FC;
   // GBK_TO_UNICODE[1137] := 16#51D5;
   // GBK_TO_UNICODE[1138] := 16#83FD;
   // GBK_TO_UNICODE[1139] := 16#51D6;
   // GBK_TO_UNICODE[1140] := 16#83FE;
   // GBK_TO_UNICODE[1141] := 16#51D7;
   // GBK_TO_UNICODE[1142] := 16#8440;
   // GBK_TO_UNICODE[1143] := 16#51D8;
   // GBK_TO_UNICODE[1144] := 16#8441;
   // GBK_TO_UNICODE[1145] := 16#51D9;
   // GBK_TO_UNICODE[1146] := 16#8442;
   // GBK_TO_UNICODE[1147] := 16#51DA;
   // GBK_TO_UNICODE[1148] := 16#8443;
   // GBK_TO_UNICODE[1149] := 16#51DC;
   // GBK_TO_UNICODE[1150] := 16#8444;
   // GBK_TO_UNICODE[1151] := 16#51DE;
   // GBK_TO_UNICODE[1152] := 16#8445;
   // GBK_TO_UNICODE[1153] := 16#51DF;
   // GBK_TO_UNICODE[1154] := 16#8446;
   // GBK_TO_UNICODE[1155] := 16#51E2;
   // GBK_TO_UNICODE[1156] := 16#8447;
   // GBK_TO_UNICODE[1157] := 16#51E3;
   // GBK_TO_UNICODE[1158] := 16#8448;
   // GBK_TO_UNICODE[1159] := 16#51E5;
   // GBK_TO_UNICODE[1160] := 16#8449;
   // GBK_TO_UNICODE[1161] := 16#51E6;
   // GBK_TO_UNICODE[1162] := 16#844A;
   // GBK_TO_UNICODE[1163] := 16#51E7;
   // GBK_TO_UNICODE[1164] := 16#844B;
   // GBK_TO_UNICODE[1165] := 16#51E8;
   // GBK_TO_UNICODE[1166] := 16#844C;
   // GBK_TO_UNICODE[1167] := 16#51E9;
   // GBK_TO_UNICODE[1168] := 16#844D;
   // GBK_TO_UNICODE[1169] := 16#51EA;
   // GBK_TO_UNICODE[1170] := 16#844E;
   // GBK_TO_UNICODE[1171] := 16#51EC;
   // GBK_TO_UNICODE[1172] := 16#844F;
   // GBK_TO_UNICODE[1173] := 16#51EE;
   // GBK_TO_UNICODE[1174] := 16#8450;
   // GBK_TO_UNICODE[1175] := 16#51F1;
   // GBK_TO_UNICODE[1176] := 16#8451;
   // GBK_TO_UNICODE[1177] := 16#51F2;
   // GBK_TO_UNICODE[1178] := 16#8452;
   // GBK_TO_UNICODE[1179] := 16#51F4;
   // GBK_TO_UNICODE[1180] := 16#8453;
   // GBK_TO_UNICODE[1181] := 16#51F7;
   // GBK_TO_UNICODE[1182] := 16#8454;
   // GBK_TO_UNICODE[1183] := 16#51FE;
   // GBK_TO_UNICODE[1184] := 16#8455;
   // GBK_TO_UNICODE[1185] := 16#5204;
   // GBK_TO_UNICODE[1186] := 16#8456;
   // GBK_TO_UNICODE[1187] := 16#5205;
   // GBK_TO_UNICODE[1188] := 16#8457;
   // GBK_TO_UNICODE[1189] := 16#5209;
   // GBK_TO_UNICODE[1190] := 16#8458;
   // GBK_TO_UNICODE[1191] := 16#520B;
   // GBK_TO_UNICODE[1192] := 16#8459;
   // GBK_TO_UNICODE[1193] := 16#520C;
   // GBK_TO_UNICODE[1194] := 16#845A;
   // GBK_TO_UNICODE[1195] := 16#520F;
   // GBK_TO_UNICODE[1196] := 16#845B;
   // GBK_TO_UNICODE[1197] := 16#5210;
   // GBK_TO_UNICODE[1198] := 16#845C;
   // GBK_TO_UNICODE[1199] := 16#5213;
   // GBK_TO_UNICODE[1200] := 16#845D;
   // GBK_TO_UNICODE[1201] := 16#5214;
   // GBK_TO_UNICODE[1202] := 16#845E;
   // GBK_TO_UNICODE[1203] := 16#5215;
   // GBK_TO_UNICODE[1204] := 16#845F;
   // GBK_TO_UNICODE[1205] := 16#521C;
   // GBK_TO_UNICODE[1206] := 16#8460;
   // GBK_TO_UNICODE[1207] := 16#521E;
   // GBK_TO_UNICODE[1208] := 16#8461;
   // GBK_TO_UNICODE[1209] := 16#521F;
   // GBK_TO_UNICODE[1210] := 16#8462;
   // GBK_TO_UNICODE[1211] := 16#5221;
   // GBK_TO_UNICODE[1212] := 16#8463;
   // GBK_TO_UNICODE[1213] := 16#5222;
   // GBK_TO_UNICODE[1214] := 16#8464;
   // GBK_TO_UNICODE[1215] := 16#5223;
   // GBK_TO_UNICODE[1216] := 16#8465;
   // GBK_TO_UNICODE[1217] := 16#5225;
   // GBK_TO_UNICODE[1218] := 16#8466;
   // GBK_TO_UNICODE[1219] := 16#5226;
   // GBK_TO_UNICODE[1220] := 16#8467;
   // GBK_TO_UNICODE[1221] := 16#5227;
   // GBK_TO_UNICODE[1222] := 16#8468;
   // GBK_TO_UNICODE[1223] := 16#522A;
   // GBK_TO_UNICODE[1224] := 16#8469;
   // GBK_TO_UNICODE[1225] := 16#522C;
   // GBK_TO_UNICODE[1226] := 16#846A;
   // GBK_TO_UNICODE[1227] := 16#522F;
   // GBK_TO_UNICODE[1228] := 16#846B;
   // GBK_TO_UNICODE[1229] := 16#5231;
   // GBK_TO_UNICODE[1230] := 16#846C;
   // GBK_TO_UNICODE[1231] := 16#5232;
   // GBK_TO_UNICODE[1232] := 16#846D;
   // GBK_TO_UNICODE[1233] := 16#5234;
   // GBK_TO_UNICODE[1234] := 16#846E;
   // GBK_TO_UNICODE[1235] := 16#5235;
   // GBK_TO_UNICODE[1236] := 16#846F;
   // GBK_TO_UNICODE[1237] := 16#523C;
   // GBK_TO_UNICODE[1238] := 16#8470;
   // GBK_TO_UNICODE[1239] := 16#523E;
   // GBK_TO_UNICODE[1240] := 16#8471;
   // GBK_TO_UNICODE[1241] := 16#5244;
   // GBK_TO_UNICODE[1242] := 16#8472;
   // GBK_TO_UNICODE[1243] := 16#5245;
   // GBK_TO_UNICODE[1244] := 16#8473;
   // GBK_TO_UNICODE[1245] := 16#5246;
   // GBK_TO_UNICODE[1246] := 16#8474;
   // GBK_TO_UNICODE[1247] := 16#5247;
   // GBK_TO_UNICODE[1248] := 16#8475;
   // GBK_TO_UNICODE[1249] := 16#5248;
   // GBK_TO_UNICODE[1250] := 16#8476;
   // GBK_TO_UNICODE[1251] := 16#5249;
   // GBK_TO_UNICODE[1252] := 16#8477;
   // GBK_TO_UNICODE[1253] := 16#524B;
   // GBK_TO_UNICODE[1254] := 16#8478;
   // GBK_TO_UNICODE[1255] := 16#524E;
   // GBK_TO_UNICODE[1256] := 16#8479;
   // GBK_TO_UNICODE[1257] := 16#524F;
   // GBK_TO_UNICODE[1258] := 16#847A;
   // GBK_TO_UNICODE[1259] := 16#5252;
   // GBK_TO_UNICODE[1260] := 16#847B;
   // GBK_TO_UNICODE[1261] := 16#5253;
   // GBK_TO_UNICODE[1262] := 16#847C;
   // GBK_TO_UNICODE[1263] := 16#5255;
   // GBK_TO_UNICODE[1264] := 16#847D;
   // GBK_TO_UNICODE[1265] := 16#5257;
   // GBK_TO_UNICODE[1266] := 16#847E;
   // GBK_TO_UNICODE[1267] := 16#5258;
   // GBK_TO_UNICODE[1268] := 16#8480;
   // GBK_TO_UNICODE[1269] := 16#5259;
   // GBK_TO_UNICODE[1270] := 16#8481;
   // GBK_TO_UNICODE[1271] := 16#525A;
   // GBK_TO_UNICODE[1272] := 16#8482;
   // GBK_TO_UNICODE[1273] := 16#525B;
   // GBK_TO_UNICODE[1274] := 16#8483;
   // GBK_TO_UNICODE[1275] := 16#525D;
   // GBK_TO_UNICODE[1276] := 16#8484;
   // GBK_TO_UNICODE[1277] := 16#525F;
   // GBK_TO_UNICODE[1278] := 16#8485;
   // GBK_TO_UNICODE[1279] := 16#5260;
   // GBK_TO_UNICODE[1280] := 16#8486;
   // GBK_TO_UNICODE[1281] := 16#5262;
   // GBK_TO_UNICODE[1282] := 16#8487;
   // GBK_TO_UNICODE[1283] := 16#5263;
   // GBK_TO_UNICODE[1284] := 16#8488;
   // GBK_TO_UNICODE[1285] := 16#5264;
   // GBK_TO_UNICODE[1286] := 16#8489;
   // GBK_TO_UNICODE[1287] := 16#5266;
   // GBK_TO_UNICODE[1288] := 16#848A;
   // GBK_TO_UNICODE[1289] := 16#5268;
   // GBK_TO_UNICODE[1290] := 16#848B;
   // GBK_TO_UNICODE[1291] := 16#526B;
   // GBK_TO_UNICODE[1292] := 16#848C;
   // GBK_TO_UNICODE[1293] := 16#526C;
   // GBK_TO_UNICODE[1294] := 16#848D;
   // GBK_TO_UNICODE[1295] := 16#526D;
   // GBK_TO_UNICODE[1296] := 16#848E;
   // GBK_TO_UNICODE[1297] := 16#526E;
   // GBK_TO_UNICODE[1298] := 16#848F;
   // GBK_TO_UNICODE[1299] := 16#5270;
   // GBK_TO_UNICODE[1300] := 16#8490;
   // GBK_TO_UNICODE[1301] := 16#5271;
   // GBK_TO_UNICODE[1302] := 16#8491;
   // GBK_TO_UNICODE[1303] := 16#5273;
   // GBK_TO_UNICODE[1304] := 16#8492;
   // GBK_TO_UNICODE[1305] := 16#5274;
   // GBK_TO_UNICODE[1306] := 16#8493;
   // GBK_TO_UNICODE[1307] := 16#5275;
   // GBK_TO_UNICODE[1308] := 16#8494;
   // GBK_TO_UNICODE[1309] := 16#5276;
   // GBK_TO_UNICODE[1310] := 16#8495;
   // GBK_TO_UNICODE[1311] := 16#5277;
   // GBK_TO_UNICODE[1312] := 16#8496;
   // GBK_TO_UNICODE[1313] := 16#5278;
   // GBK_TO_UNICODE[1314] := 16#8497;
   // GBK_TO_UNICODE[1315] := 16#5279;
   // GBK_TO_UNICODE[1316] := 16#8498;
   // GBK_TO_UNICODE[1317] := 16#527A;
   // GBK_TO_UNICODE[1318] := 16#8499;
   // GBK_TO_UNICODE[1319] := 16#527B;
   // GBK_TO_UNICODE[1320] := 16#849A;
   // GBK_TO_UNICODE[1321] := 16#527C;
   // GBK_TO_UNICODE[1322] := 16#849B;
   // GBK_TO_UNICODE[1323] := 16#527E;
   // GBK_TO_UNICODE[1324] := 16#849C;
   // GBK_TO_UNICODE[1325] := 16#5280;
   // GBK_TO_UNICODE[1326] := 16#849D;
   // GBK_TO_UNICODE[1327] := 16#5283;
   // GBK_TO_UNICODE[1328] := 16#849E;
   // GBK_TO_UNICODE[1329] := 16#5284;
   // GBK_TO_UNICODE[1330] := 16#849F;
   // GBK_TO_UNICODE[1331] := 16#5285;
   // GBK_TO_UNICODE[1332] := 16#84A0;
   // GBK_TO_UNICODE[1333] := 16#5286;
   // GBK_TO_UNICODE[1334] := 16#84A1;
   // GBK_TO_UNICODE[1335] := 16#5287;
   // GBK_TO_UNICODE[1336] := 16#84A2;
   // GBK_TO_UNICODE[1337] := 16#5289;
   // GBK_TO_UNICODE[1338] := 16#84A3;
   // GBK_TO_UNICODE[1339] := 16#528A;
   // GBK_TO_UNICODE[1340] := 16#84A4;
   // GBK_TO_UNICODE[1341] := 16#528B;
   // GBK_TO_UNICODE[1342] := 16#84A5;
   // GBK_TO_UNICODE[1343] := 16#528C;
   // GBK_TO_UNICODE[1344] := 16#84A6;
   // GBK_TO_UNICODE[1345] := 16#528D;
   // GBK_TO_UNICODE[1346] := 16#84A7;
   // GBK_TO_UNICODE[1347] := 16#528E;
   // GBK_TO_UNICODE[1348] := 16#84A8;
   // GBK_TO_UNICODE[1349] := 16#528F;
   // GBK_TO_UNICODE[1350] := 16#84A9;
   // GBK_TO_UNICODE[1351] := 16#5291;
   // GBK_TO_UNICODE[1352] := 16#84AA;
   // GBK_TO_UNICODE[1353] := 16#5292;
   // GBK_TO_UNICODE[1354] := 16#84AB;
   // GBK_TO_UNICODE[1355] := 16#5294;
   // GBK_TO_UNICODE[1356] := 16#84AC;
   // GBK_TO_UNICODE[1357] := 16#5295;
   // GBK_TO_UNICODE[1358] := 16#84AD;
   // GBK_TO_UNICODE[1359] := 16#5296;
   // GBK_TO_UNICODE[1360] := 16#84AE;
   // GBK_TO_UNICODE[1361] := 16#5297;
   // GBK_TO_UNICODE[1362] := 16#84AF;
   // GBK_TO_UNICODE[1363] := 16#5298;
   // GBK_TO_UNICODE[1364] := 16#84B0;
   // GBK_TO_UNICODE[1365] := 16#5299;
   // GBK_TO_UNICODE[1366] := 16#84B1;
   // GBK_TO_UNICODE[1367] := 16#529A;
   // GBK_TO_UNICODE[1368] := 16#84B2;
   // GBK_TO_UNICODE[1369] := 16#529C;
   // GBK_TO_UNICODE[1370] := 16#84B3;
   // GBK_TO_UNICODE[1371] := 16#52A4;
   // GBK_TO_UNICODE[1372] := 16#84B4;
   // GBK_TO_UNICODE[1373] := 16#52A5;
   // GBK_TO_UNICODE[1374] := 16#84B5;
   // GBK_TO_UNICODE[1375] := 16#52A6;
   // GBK_TO_UNICODE[1376] := 16#84B6;
   // GBK_TO_UNICODE[1377] := 16#52A7;
   // GBK_TO_UNICODE[1378] := 16#84B7;
   // GBK_TO_UNICODE[1379] := 16#52AE;
   // GBK_TO_UNICODE[1380] := 16#84B8;
   // GBK_TO_UNICODE[1381] := 16#52AF;
   // GBK_TO_UNICODE[1382] := 16#84B9;
   // GBK_TO_UNICODE[1383] := 16#52B0;
   // GBK_TO_UNICODE[1384] := 16#84BA;
   // GBK_TO_UNICODE[1385] := 16#52B4;
   // GBK_TO_UNICODE[1386] := 16#84BB;
   // GBK_TO_UNICODE[1387] := 16#52B5;
   // GBK_TO_UNICODE[1388] := 16#84BC;
   // GBK_TO_UNICODE[1389] := 16#52B6;
   // GBK_TO_UNICODE[1390] := 16#84BD;
   // GBK_TO_UNICODE[1391] := 16#52B7;
   // GBK_TO_UNICODE[1392] := 16#84BE;
   // GBK_TO_UNICODE[1393] := 16#52B8;
   // GBK_TO_UNICODE[1394] := 16#84BF;
   // GBK_TO_UNICODE[1395] := 16#52B9;
   // GBK_TO_UNICODE[1396] := 16#84C0;
   // GBK_TO_UNICODE[1397] := 16#52BA;
   // GBK_TO_UNICODE[1398] := 16#84C1;
   // GBK_TO_UNICODE[1399] := 16#52BB;
   // GBK_TO_UNICODE[1400] := 16#84C2;
   // GBK_TO_UNICODE[1401] := 16#52BC;
   // GBK_TO_UNICODE[1402] := 16#84C3;
   // GBK_TO_UNICODE[1403] := 16#52BD;
   // GBK_TO_UNICODE[1404] := 16#84C4;
   // GBK_TO_UNICODE[1405] := 16#52C0;
   // GBK_TO_UNICODE[1406] := 16#84C5;
   // GBK_TO_UNICODE[1407] := 16#52C1;
   // GBK_TO_UNICODE[1408] := 16#84C6;
   // GBK_TO_UNICODE[1409] := 16#52C2;
   // GBK_TO_UNICODE[1410] := 16#84C7;
   // GBK_TO_UNICODE[1411] := 16#52C4;
   // GBK_TO_UNICODE[1412] := 16#84C8;
   // GBK_TO_UNICODE[1413] := 16#52C5;
   // GBK_TO_UNICODE[1414] := 16#84C9;
   // GBK_TO_UNICODE[1415] := 16#52C6;
   // GBK_TO_UNICODE[1416] := 16#84CA;
   // GBK_TO_UNICODE[1417] := 16#52C8;
   // GBK_TO_UNICODE[1418] := 16#84CB;
   // GBK_TO_UNICODE[1419] := 16#52CA;
   // GBK_TO_UNICODE[1420] := 16#84CC;
   // GBK_TO_UNICODE[1421] := 16#52CC;
   // GBK_TO_UNICODE[1422] := 16#84CD;
   // GBK_TO_UNICODE[1423] := 16#52CD;
   // GBK_TO_UNICODE[1424] := 16#84CE;
   // GBK_TO_UNICODE[1425] := 16#52CE;
   // GBK_TO_UNICODE[1426] := 16#84CF;
   // GBK_TO_UNICODE[1427] := 16#52CF;
   // GBK_TO_UNICODE[1428] := 16#84D0;
   // GBK_TO_UNICODE[1429] := 16#52D1;
   // GBK_TO_UNICODE[1430] := 16#84D1;
   // GBK_TO_UNICODE[1431] := 16#52D3;
   // GBK_TO_UNICODE[1432] := 16#84D2;
   // GBK_TO_UNICODE[1433] := 16#52D4;
   // GBK_TO_UNICODE[1434] := 16#84D3;
   // GBK_TO_UNICODE[1435] := 16#52D5;
   // GBK_TO_UNICODE[1436] := 16#84D4;
   // GBK_TO_UNICODE[1437] := 16#52D7;
   // GBK_TO_UNICODE[1438] := 16#84D5;
   // GBK_TO_UNICODE[1439] := 16#52D9;
   // GBK_TO_UNICODE[1440] := 16#84D6;
   // GBK_TO_UNICODE[1441] := 16#52DA;
   // GBK_TO_UNICODE[1442] := 16#84D7;
   // GBK_TO_UNICODE[1443] := 16#52DB;
   // GBK_TO_UNICODE[1444] := 16#84D8;
   // GBK_TO_UNICODE[1445] := 16#52DC;
   // GBK_TO_UNICODE[1446] := 16#84D9;
   // GBK_TO_UNICODE[1447] := 16#52DD;
   // GBK_TO_UNICODE[1448] := 16#84DA;
   // GBK_TO_UNICODE[1449] := 16#52DE;
   // GBK_TO_UNICODE[1450] := 16#84DB;
   // GBK_TO_UNICODE[1451] := 16#52E0;
   // GBK_TO_UNICODE[1452] := 16#84DC;
   // GBK_TO_UNICODE[1453] := 16#52E1;
   // GBK_TO_UNICODE[1454] := 16#84DD;
   // GBK_TO_UNICODE[1455] := 16#52E2;
   // GBK_TO_UNICODE[1456] := 16#84DE;
   // GBK_TO_UNICODE[1457] := 16#52E3;
   // GBK_TO_UNICODE[1458] := 16#84DF;
   // GBK_TO_UNICODE[1459] := 16#52E5;
   // GBK_TO_UNICODE[1460] := 16#84E0;
   // GBK_TO_UNICODE[1461] := 16#52E6;
   // GBK_TO_UNICODE[1462] := 16#84E1;
   // GBK_TO_UNICODE[1463] := 16#52E7;
   // GBK_TO_UNICODE[1464] := 16#84E2;
   // GBK_TO_UNICODE[1465] := 16#52E8;
   // GBK_TO_UNICODE[1466] := 16#84E3;
   // GBK_TO_UNICODE[1467] := 16#52E9;
   // GBK_TO_UNICODE[1468] := 16#84E4;
   // GBK_TO_UNICODE[1469] := 16#52EA;
   // GBK_TO_UNICODE[1470] := 16#84E5;
   // GBK_TO_UNICODE[1471] := 16#52EB;
   // GBK_TO_UNICODE[1472] := 16#84E6;
   // GBK_TO_UNICODE[1473] := 16#52EC;
   // GBK_TO_UNICODE[1474] := 16#84E7;
   // GBK_TO_UNICODE[1475] := 16#52ED;
   // GBK_TO_UNICODE[1476] := 16#84E8;
   // GBK_TO_UNICODE[1477] := 16#52EE;
   // GBK_TO_UNICODE[1478] := 16#84E9;
   // GBK_TO_UNICODE[1479] := 16#52EF;
   // GBK_TO_UNICODE[1480] := 16#84EA;
   // GBK_TO_UNICODE[1481] := 16#52F1;
   // GBK_TO_UNICODE[1482] := 16#84EB;
   // GBK_TO_UNICODE[1483] := 16#52F2;
   // GBK_TO_UNICODE[1484] := 16#84EC;
   // GBK_TO_UNICODE[1485] := 16#52F3;
   // GBK_TO_UNICODE[1486] := 16#84ED;
   // GBK_TO_UNICODE[1487] := 16#52F4;
   // GBK_TO_UNICODE[1488] := 16#84EE;
   // GBK_TO_UNICODE[1489] := 16#52F5;
   // GBK_TO_UNICODE[1490] := 16#84EF;
   // GBK_TO_UNICODE[1491] := 16#52F6;
   // GBK_TO_UNICODE[1492] := 16#84F0;
   // GBK_TO_UNICODE[1493] := 16#52F7;
   // GBK_TO_UNICODE[1494] := 16#84F1;
   // GBK_TO_UNICODE[1495] := 16#52F8;
   // GBK_TO_UNICODE[1496] := 16#84F2;
   // GBK_TO_UNICODE[1497] := 16#52FB;
   // GBK_TO_UNICODE[1498] := 16#84F3;
   // GBK_TO_UNICODE[1499] := 16#52FC;
   // GBK_TO_UNICODE[1500] := 16#84F4;
   // GBK_TO_UNICODE[1501] := 16#52FD;
   // GBK_TO_UNICODE[1502] := 16#84F5;
   // GBK_TO_UNICODE[1503] := 16#5301;
   // GBK_TO_UNICODE[1504] := 16#84F6;
   // GBK_TO_UNICODE[1505] := 16#5302;
   // GBK_TO_UNICODE[1506] := 16#84F7;
   // GBK_TO_UNICODE[1507] := 16#5303;
   // GBK_TO_UNICODE[1508] := 16#84F8;
   // GBK_TO_UNICODE[1509] := 16#5304;
   // GBK_TO_UNICODE[1510] := 16#84F9;
   // GBK_TO_UNICODE[1511] := 16#5307;
   // GBK_TO_UNICODE[1512] := 16#84FA;
   // GBK_TO_UNICODE[1513] := 16#5309;
   // GBK_TO_UNICODE[1514] := 16#84FB;
   // GBK_TO_UNICODE[1515] := 16#530A;
   // GBK_TO_UNICODE[1516] := 16#84FC;
   // GBK_TO_UNICODE[1517] := 16#530B;
   // GBK_TO_UNICODE[1518] := 16#84FD;
   // GBK_TO_UNICODE[1519] := 16#530C;
   // GBK_TO_UNICODE[1520] := 16#84FE;
   // GBK_TO_UNICODE[1521] := 16#530E;
   // GBK_TO_UNICODE[1522] := 16#8540;
   // GBK_TO_UNICODE[1523] := 16#5311;
   // GBK_TO_UNICODE[1524] := 16#8541;
   // GBK_TO_UNICODE[1525] := 16#5312;
   // GBK_TO_UNICODE[1526] := 16#8542;
   // GBK_TO_UNICODE[1527] := 16#5313;
   // GBK_TO_UNICODE[1528] := 16#8543;
   // GBK_TO_UNICODE[1529] := 16#5314;
   // GBK_TO_UNICODE[1530] := 16#8544;
   // GBK_TO_UNICODE[1531] := 16#5318;
   // GBK_TO_UNICODE[1532] := 16#8545;
   // GBK_TO_UNICODE[1533] := 16#531B;
   // GBK_TO_UNICODE[1534] := 16#8546;
   // GBK_TO_UNICODE[1535] := 16#531C;
   // GBK_TO_UNICODE[1536] := 16#8547;
   // GBK_TO_UNICODE[1537] := 16#531E;
   // GBK_TO_UNICODE[1538] := 16#8548;
   // GBK_TO_UNICODE[1539] := 16#531F;
   // GBK_TO_UNICODE[1540] := 16#8549;
   // GBK_TO_UNICODE[1541] := 16#5322;
   // GBK_TO_UNICODE[1542] := 16#854A;
   // GBK_TO_UNICODE[1543] := 16#5324;
   // GBK_TO_UNICODE[1544] := 16#854B;
   // GBK_TO_UNICODE[1545] := 16#5325;
   // GBK_TO_UNICODE[1546] := 16#854C;
   // GBK_TO_UNICODE[1547] := 16#5327;
   // GBK_TO_UNICODE[1548] := 16#854D;
   // GBK_TO_UNICODE[1549] := 16#5328;
   // GBK_TO_UNICODE[1550] := 16#854E;
   // GBK_TO_UNICODE[1551] := 16#5329;
   // GBK_TO_UNICODE[1552] := 16#854F;
   // GBK_TO_UNICODE[1553] := 16#532B;
   // GBK_TO_UNICODE[1554] := 16#8550;
   // GBK_TO_UNICODE[1555] := 16#532C;
   // GBK_TO_UNICODE[1556] := 16#8551;
   // GBK_TO_UNICODE[1557] := 16#532D;
   // GBK_TO_UNICODE[1558] := 16#8552;
   // GBK_TO_UNICODE[1559] := 16#532F;
   // GBK_TO_UNICODE[1560] := 16#8553;
   // GBK_TO_UNICODE[1561] := 16#5330;
   // GBK_TO_UNICODE[1562] := 16#8554;
   // GBK_TO_UNICODE[1563] := 16#5331;
   // GBK_TO_UNICODE[1564] := 16#8555;
   // GBK_TO_UNICODE[1565] := 16#5332;
   // GBK_TO_UNICODE[1566] := 16#8556;
   // GBK_TO_UNICODE[1567] := 16#5333;
   // GBK_TO_UNICODE[1568] := 16#8557;
   // GBK_TO_UNICODE[1569] := 16#5334;
   // GBK_TO_UNICODE[1570] := 16#8558;
   // GBK_TO_UNICODE[1571] := 16#5335;
   // GBK_TO_UNICODE[1572] := 16#8559;
   // GBK_TO_UNICODE[1573] := 16#5336;
   // GBK_TO_UNICODE[1574] := 16#855A;
   // GBK_TO_UNICODE[1575] := 16#5337;
   // GBK_TO_UNICODE[1576] := 16#855B;
   // GBK_TO_UNICODE[1577] := 16#5338;
   // GBK_TO_UNICODE[1578] := 16#855C;
   // GBK_TO_UNICODE[1579] := 16#533C;
   // GBK_TO_UNICODE[1580] := 16#855D;
   // GBK_TO_UNICODE[1581] := 16#533D;
   // GBK_TO_UNICODE[1582] := 16#855E;
   // GBK_TO_UNICODE[1583] := 16#5340;
   // GBK_TO_UNICODE[1584] := 16#855F;
   // GBK_TO_UNICODE[1585] := 16#5342;
   // GBK_TO_UNICODE[1586] := 16#8560;
   // GBK_TO_UNICODE[1587] := 16#5344;
   // GBK_TO_UNICODE[1588] := 16#8561;
   // GBK_TO_UNICODE[1589] := 16#5346;
   // GBK_TO_UNICODE[1590] := 16#8562;
   // GBK_TO_UNICODE[1591] := 16#534B;
   // GBK_TO_UNICODE[1592] := 16#8563;
   // GBK_TO_UNICODE[1593] := 16#534C;
   // GBK_TO_UNICODE[1594] := 16#8564;
   // GBK_TO_UNICODE[1595] := 16#534D;
   // GBK_TO_UNICODE[1596] := 16#8565;
   // GBK_TO_UNICODE[1597] := 16#5350;
   // GBK_TO_UNICODE[1598] := 16#8566;
   // GBK_TO_UNICODE[1599] := 16#5354;
   // GBK_TO_UNICODE[1600] := 16#8567;
   // GBK_TO_UNICODE[1601] := 16#5358;
   // GBK_TO_UNICODE[1602] := 16#8568;
   // GBK_TO_UNICODE[1603] := 16#5359;
   // GBK_TO_UNICODE[1604] := 16#8569;
   // GBK_TO_UNICODE[1605] := 16#535B;
   // GBK_TO_UNICODE[1606] := 16#856A;
   // GBK_TO_UNICODE[1607] := 16#535D;
   // GBK_TO_UNICODE[1608] := 16#856B;
   // GBK_TO_UNICODE[1609] := 16#5365;
   // GBK_TO_UNICODE[1610] := 16#856C;
   // GBK_TO_UNICODE[1611] := 16#5368;
   // GBK_TO_UNICODE[1612] := 16#856D;
   // GBK_TO_UNICODE[1613] := 16#536A;
   // GBK_TO_UNICODE[1614] := 16#856E;
   // GBK_TO_UNICODE[1615] := 16#536C;
   // GBK_TO_UNICODE[1616] := 16#856F;
   // GBK_TO_UNICODE[1617] := 16#536D;
   // GBK_TO_UNICODE[1618] := 16#8570;
   // GBK_TO_UNICODE[1619] := 16#5372;
   // GBK_TO_UNICODE[1620] := 16#8571;
   // GBK_TO_UNICODE[1621] := 16#5376;
   // GBK_TO_UNICODE[1622] := 16#8572;
   // GBK_TO_UNICODE[1623] := 16#5379;
   // GBK_TO_UNICODE[1624] := 16#8573;
   // GBK_TO_UNICODE[1625] := 16#537B;
   // GBK_TO_UNICODE[1626] := 16#8574;
   // GBK_TO_UNICODE[1627] := 16#537C;
   // GBK_TO_UNICODE[1628] := 16#8575;
   // GBK_TO_UNICODE[1629] := 16#537D;
   // GBK_TO_UNICODE[1630] := 16#8576;
   // GBK_TO_UNICODE[1631] := 16#537E;
   // GBK_TO_UNICODE[1632] := 16#8577;
   // GBK_TO_UNICODE[1633] := 16#5380;
   // GBK_TO_UNICODE[1634] := 16#8578;
   // GBK_TO_UNICODE[1635] := 16#5381;
   // GBK_TO_UNICODE[1636] := 16#8579;
   // GBK_TO_UNICODE[1637] := 16#5383;
   // GBK_TO_UNICODE[1638] := 16#857A;
   // GBK_TO_UNICODE[1639] := 16#5387;
   // GBK_TO_UNICODE[1640] := 16#857B;
   // GBK_TO_UNICODE[1641] := 16#5388;
   // GBK_TO_UNICODE[1642] := 16#857C;
   // GBK_TO_UNICODE[1643] := 16#538A;
   // GBK_TO_UNICODE[1644] := 16#857D;
   // GBK_TO_UNICODE[1645] := 16#538E;
   // GBK_TO_UNICODE[1646] := 16#857E;
   // GBK_TO_UNICODE[1647] := 16#538F;
   // GBK_TO_UNICODE[1648] := 16#8580;
   // GBK_TO_UNICODE[1649] := 16#5390;
   // GBK_TO_UNICODE[1650] := 16#8581;
   // GBK_TO_UNICODE[1651] := 16#5391;
   // GBK_TO_UNICODE[1652] := 16#8582;
   // GBK_TO_UNICODE[1653] := 16#5392;
   // GBK_TO_UNICODE[1654] := 16#8583;
   // GBK_TO_UNICODE[1655] := 16#5393;
   // GBK_TO_UNICODE[1656] := 16#8584;
   // GBK_TO_UNICODE[1657] := 16#5394;
   // GBK_TO_UNICODE[1658] := 16#8585;
   // GBK_TO_UNICODE[1659] := 16#5396;
   // GBK_TO_UNICODE[1660] := 16#8586;
   // GBK_TO_UNICODE[1661] := 16#5397;
   // GBK_TO_UNICODE[1662] := 16#8587;
   // GBK_TO_UNICODE[1663] := 16#5399;
   // GBK_TO_UNICODE[1664] := 16#8588;
   // GBK_TO_UNICODE[1665] := 16#539B;
   // GBK_TO_UNICODE[1666] := 16#8589;
   // GBK_TO_UNICODE[1667] := 16#539C;
   // GBK_TO_UNICODE[1668] := 16#858A;
   // GBK_TO_UNICODE[1669] := 16#539E;
   // GBK_TO_UNICODE[1670] := 16#858B;
   // GBK_TO_UNICODE[1671] := 16#53A0;
   // GBK_TO_UNICODE[1672] := 16#858C;
   // GBK_TO_UNICODE[1673] := 16#53A1;
   // GBK_TO_UNICODE[1674] := 16#858D;
   // GBK_TO_UNICODE[1675] := 16#53A4;
   // GBK_TO_UNICODE[1676] := 16#858E;
   // GBK_TO_UNICODE[1677] := 16#53A7;
   // GBK_TO_UNICODE[1678] := 16#858F;
   // GBK_TO_UNICODE[1679] := 16#53AA;
   // GBK_TO_UNICODE[1680] := 16#8590;
   // GBK_TO_UNICODE[1681] := 16#53AB;
   // GBK_TO_UNICODE[1682] := 16#8591;
   // GBK_TO_UNICODE[1683] := 16#53AC;
   // GBK_TO_UNICODE[1684] := 16#8592;
   // GBK_TO_UNICODE[1685] := 16#53AD;
   // GBK_TO_UNICODE[1686] := 16#8593;
   // GBK_TO_UNICODE[1687] := 16#53AF;
   // GBK_TO_UNICODE[1688] := 16#8594;
   // GBK_TO_UNICODE[1689] := 16#53B0;
   // GBK_TO_UNICODE[1690] := 16#8595;
   // GBK_TO_UNICODE[1691] := 16#53B1;
   // GBK_TO_UNICODE[1692] := 16#8596;
   // GBK_TO_UNICODE[1693] := 16#53B2;
   // GBK_TO_UNICODE[1694] := 16#8597;
   // GBK_TO_UNICODE[1695] := 16#53B3;
   // GBK_TO_UNICODE[1696] := 16#8598;
   // GBK_TO_UNICODE[1697] := 16#53B4;
   // GBK_TO_UNICODE[1698] := 16#8599;
   // GBK_TO_UNICODE[1699] := 16#53B5;
   // GBK_TO_UNICODE[1700] := 16#859A;
   // GBK_TO_UNICODE[1701] := 16#53B7;
   // GBK_TO_UNICODE[1702] := 16#859B;
   // GBK_TO_UNICODE[1703] := 16#53B8;
   // GBK_TO_UNICODE[1704] := 16#859C;
   // GBK_TO_UNICODE[1705] := 16#53B9;
   // GBK_TO_UNICODE[1706] := 16#859D;
   // GBK_TO_UNICODE[1707] := 16#53BA;
   // GBK_TO_UNICODE[1708] := 16#859E;
   // GBK_TO_UNICODE[1709] := 16#53BC;
   // GBK_TO_UNICODE[1710] := 16#859F;
   // GBK_TO_UNICODE[1711] := 16#53BD;
   // GBK_TO_UNICODE[1712] := 16#85A0;
   // GBK_TO_UNICODE[1713] := 16#53BE;
   // GBK_TO_UNICODE[1714] := 16#85A1;
   // GBK_TO_UNICODE[1715] := 16#53C0;
   // GBK_TO_UNICODE[1716] := 16#85A2;
   // GBK_TO_UNICODE[1717] := 16#53C3;
   // GBK_TO_UNICODE[1718] := 16#85A3;
   // GBK_TO_UNICODE[1719] := 16#53C4;
   // GBK_TO_UNICODE[1720] := 16#85A4;
   // GBK_TO_UNICODE[1721] := 16#53C5;
   // GBK_TO_UNICODE[1722] := 16#85A5;
   // GBK_TO_UNICODE[1723] := 16#53C6;
   // GBK_TO_UNICODE[1724] := 16#85A6;
   // GBK_TO_UNICODE[1725] := 16#53C7;
   // GBK_TO_UNICODE[1726] := 16#85A7;
   // GBK_TO_UNICODE[1727] := 16#53CE;
   // GBK_TO_UNICODE[1728] := 16#85A8;
   // GBK_TO_UNICODE[1729] := 16#53CF;
   // GBK_TO_UNICODE[1730] := 16#85A9;
   // GBK_TO_UNICODE[1731] := 16#53D0;
   // GBK_TO_UNICODE[1732] := 16#85AA;
   // GBK_TO_UNICODE[1733] := 16#53D2;
   // GBK_TO_UNICODE[1734] := 16#85AB;
   // GBK_TO_UNICODE[1735] := 16#53D3;
   // GBK_TO_UNICODE[1736] := 16#85AC;
   // GBK_TO_UNICODE[1737] := 16#53D5;
   // GBK_TO_UNICODE[1738] := 16#85AD;
   // GBK_TO_UNICODE[1739] := 16#53DA;
   // GBK_TO_UNICODE[1740] := 16#85AE;
   // GBK_TO_UNICODE[1741] := 16#53DC;
   // GBK_TO_UNICODE[1742] := 16#85AF;
   // GBK_TO_UNICODE[1743] := 16#53DD;
   // GBK_TO_UNICODE[1744] := 16#85B0;
   // GBK_TO_UNICODE[1745] := 16#53DE;
   // GBK_TO_UNICODE[1746] := 16#85B1;
   // GBK_TO_UNICODE[1747] := 16#53E1;
   // GBK_TO_UNICODE[1748] := 16#85B2;
   // GBK_TO_UNICODE[1749] := 16#53E2;
   // GBK_TO_UNICODE[1750] := 16#85B3;
   // GBK_TO_UNICODE[1751] := 16#53E7;
   // GBK_TO_UNICODE[1752] := 16#85B4;
   // GBK_TO_UNICODE[1753] := 16#53F4;
   // GBK_TO_UNICODE[1754] := 16#85B5;
   // GBK_TO_UNICODE[1755] := 16#53FA;
   // GBK_TO_UNICODE[1756] := 16#85B6;
   // GBK_TO_UNICODE[1757] := 16#53FE;
   // GBK_TO_UNICODE[1758] := 16#85B7;
   // GBK_TO_UNICODE[1759] := 16#53FF;
   // GBK_TO_UNICODE[1760] := 16#85B8;
   // GBK_TO_UNICODE[1761] := 16#5400;
   // GBK_TO_UNICODE[1762] := 16#85B9;
   // GBK_TO_UNICODE[1763] := 16#5402;
   // GBK_TO_UNICODE[1764] := 16#85BA;
   // GBK_TO_UNICODE[1765] := 16#5405;
   // GBK_TO_UNICODE[1766] := 16#85BB;
   // GBK_TO_UNICODE[1767] := 16#5407;
   // GBK_TO_UNICODE[1768] := 16#85BC;
   // GBK_TO_UNICODE[1769] := 16#540B;
   // GBK_TO_UNICODE[1770] := 16#85BD;
   // GBK_TO_UNICODE[1771] := 16#5414;
   // GBK_TO_UNICODE[1772] := 16#85BE;
   // GBK_TO_UNICODE[1773] := 16#5418;
   // GBK_TO_UNICODE[1774] := 16#85BF;
   // GBK_TO_UNICODE[1775] := 16#5419;
   // GBK_TO_UNICODE[1776] := 16#85C0;
   // GBK_TO_UNICODE[1777] := 16#541A;
   // GBK_TO_UNICODE[1778] := 16#85C1;
   // GBK_TO_UNICODE[1779] := 16#541C;
   // GBK_TO_UNICODE[1780] := 16#85C2;
   // GBK_TO_UNICODE[1781] := 16#5422;
   // GBK_TO_UNICODE[1782] := 16#85C3;
   // GBK_TO_UNICODE[1783] := 16#5424;
   // GBK_TO_UNICODE[1784] := 16#85C4;
   // GBK_TO_UNICODE[1785] := 16#5425;
   // GBK_TO_UNICODE[1786] := 16#85C5;
   // GBK_TO_UNICODE[1787] := 16#542A;
   // GBK_TO_UNICODE[1788] := 16#85C6;
   // GBK_TO_UNICODE[1789] := 16#5430;
   // GBK_TO_UNICODE[1790] := 16#85C7;
   // GBK_TO_UNICODE[1791] := 16#5433;
   // GBK_TO_UNICODE[1792] := 16#85C8;
   // GBK_TO_UNICODE[1793] := 16#5436;
   // GBK_TO_UNICODE[1794] := 16#85C9;
   // GBK_TO_UNICODE[1795] := 16#5437;
   // GBK_TO_UNICODE[1796] := 16#85CA;
   // GBK_TO_UNICODE[1797] := 16#543A;
   // GBK_TO_UNICODE[1798] := 16#85CB;
   // GBK_TO_UNICODE[1799] := 16#543D;
   // GBK_TO_UNICODE[1800] := 16#85CC;
   // GBK_TO_UNICODE[1801] := 16#543F;
   // GBK_TO_UNICODE[1802] := 16#85CD;
   // GBK_TO_UNICODE[1803] := 16#5441;
   // GBK_TO_UNICODE[1804] := 16#85CE;
   // GBK_TO_UNICODE[1805] := 16#5442;
   // GBK_TO_UNICODE[1806] := 16#85CF;
   // GBK_TO_UNICODE[1807] := 16#5444;
   // GBK_TO_UNICODE[1808] := 16#85D0;
   // GBK_TO_UNICODE[1809] := 16#5445;
   // GBK_TO_UNICODE[1810] := 16#85D1;
   // GBK_TO_UNICODE[1811] := 16#5447;
   // GBK_TO_UNICODE[1812] := 16#85D2;
   // GBK_TO_UNICODE[1813] := 16#5449;
   // GBK_TO_UNICODE[1814] := 16#85D3;
   // GBK_TO_UNICODE[1815] := 16#544C;
   // GBK_TO_UNICODE[1816] := 16#85D4;
   // GBK_TO_UNICODE[1817] := 16#544D;
   // GBK_TO_UNICODE[1818] := 16#85D5;
   // GBK_TO_UNICODE[1819] := 16#544E;
   // GBK_TO_UNICODE[1820] := 16#85D6;
   // GBK_TO_UNICODE[1821] := 16#544F;
   // GBK_TO_UNICODE[1822] := 16#85D7;
   // GBK_TO_UNICODE[1823] := 16#5451;
   // GBK_TO_UNICODE[1824] := 16#85D8;
   // GBK_TO_UNICODE[1825] := 16#545A;
   // GBK_TO_UNICODE[1826] := 16#85D9;
   // GBK_TO_UNICODE[1827] := 16#545D;
   // GBK_TO_UNICODE[1828] := 16#85DA;
   // GBK_TO_UNICODE[1829] := 16#545E;
   // GBK_TO_UNICODE[1830] := 16#85DB;
   // GBK_TO_UNICODE[1831] := 16#545F;
   // GBK_TO_UNICODE[1832] := 16#85DC;
   // GBK_TO_UNICODE[1833] := 16#5460;
   // GBK_TO_UNICODE[1834] := 16#85DD;
   // GBK_TO_UNICODE[1835] := 16#5461;
   // GBK_TO_UNICODE[1836] := 16#85DE;
   // GBK_TO_UNICODE[1837] := 16#5463;
   // GBK_TO_UNICODE[1838] := 16#85DF;
   // GBK_TO_UNICODE[1839] := 16#5465;
   // GBK_TO_UNICODE[1840] := 16#85E0;
   // GBK_TO_UNICODE[1841] := 16#5467;
   // GBK_TO_UNICODE[1842] := 16#85E1;
   // GBK_TO_UNICODE[1843] := 16#5469;
   // GBK_TO_UNICODE[1844] := 16#85E2;
   // GBK_TO_UNICODE[1845] := 16#546A;
   // GBK_TO_UNICODE[1846] := 16#85E3;
   // GBK_TO_UNICODE[1847] := 16#546B;
   // GBK_TO_UNICODE[1848] := 16#85E4;
   // GBK_TO_UNICODE[1849] := 16#546C;
   // GBK_TO_UNICODE[1850] := 16#85E5;
   // GBK_TO_UNICODE[1851] := 16#546D;
   // GBK_TO_UNICODE[1852] := 16#85E6;
   // GBK_TO_UNICODE[1853] := 16#546E;
   // GBK_TO_UNICODE[1854] := 16#85E7;
   // GBK_TO_UNICODE[1855] := 16#546F;
   // GBK_TO_UNICODE[1856] := 16#85E8;
   // GBK_TO_UNICODE[1857] := 16#5470;
   // GBK_TO_UNICODE[1858] := 16#85E9;
   // GBK_TO_UNICODE[1859] := 16#5474;
   // GBK_TO_UNICODE[1860] := 16#85EA;
   // GBK_TO_UNICODE[1861] := 16#5479;
   // GBK_TO_UNICODE[1862] := 16#85EB;
   // GBK_TO_UNICODE[1863] := 16#547A;
   // GBK_TO_UNICODE[1864] := 16#85EC;
